// tc_mca_std_lib/POUs/ChangeConfig/FB_ReadParameterInNc_v1_00
///#########################################################
///Function block to read parameter in Nc.
///
///	Library:		
///	Tc2_MC2.lib
/// Tc2_System.lib
///
///	Global Variables:
///	
///	Data types:
///	
///	External functions:
///
///	History:
///	2014-02-05	v1.00	NB	Release code.
///
///	Known bugs:
///
///
///
///###########################################################
FUNCTION_BLOCK FB_ReadParameterInNc_v1_00
VAR_INPUT
	bExecute: BOOL;
	///16#4000=Axisdata, 16#5000=Encoderdata, 16#6000=Controldata, 16#7000=Drivedata
	nDeviceGroup: UDINT;
	nIndexOffset: UDINT;
END_VAR
VAR_OUTPUT
	nData: DWORD;
	bBusy: BOOL;
	bDone: BOOL;
	bError: BOOL;
	nErrorId: UDINT;
END_VAR
VAR_IN_OUT
	Axis: AXIS_REF;
END_VAR
VAR
	nState: UINT;
	fbADSREAD: ADSREAD;
END_VAR

(*Sequence to read parameter in Nc*)
CASE nState OF
0:  (*Start sequence. Wait until bExecute is TRUE*)
	IF bExecute THEN
		bBusy:=TRUE;
		bError:=FALSE;
		nErrorId:=0;
		nState:=10;
	END_IF

10: (*Read parameter in Nc*)
	fbADSREAD(
		PORT:=500,
		IDXGRP:=nDeviceGroup+Axis.NcToPlc.AxisId,
		IDXOFFS:=nIndexOffset,
		LEN:=SIZEOF(nData),
		DESTADDR:=ADR(nData),
		READ:=TRUE);

	(*Wait until it's done or if an error occurs*)
	IF NOT fbADSREAD.ERR THEN
		IF NOT fbADSREAD.BUSY THEN
			fbADSREAD(READ:=FALSE);
			nState:=20;
		END_IF
	ELSE
		nErrorId:=fbADSREAD.ERRID;
		nState:=999;
	END_IF

20: (*Sequense is done. Waits until bExecute is FALSE*)
	bBusy:=FALSE;
	bDone:=TRUE;
	IF NOT bExecute THEN
		bDone:=FALSE;
		nState:=0;
	END_IF

999: (*Error in sequence*)
	bError:=TRUE;
	bBusy:=FALSE;
	bDone:=FALSE;
	fbADSREAD(READ:=FALSE);
	IF NOT bExecute THEN
		nState:=0;
	END_IF

END_CASE

END_FUNCTION_BLOCK

// tc_mca_std_lib/POUs/Motion/Homing/FB_HomeWriteSoftLimEnable
FUNCTION_BLOCK FB_HomeWriteSoftLimEnable
VAR_INPUT
	En: BOOL;
	bReset: BOOL;
    bExecute: BOOL;		
	bSofLimEnableLow: BOOL:=TRUE;
	bSofLimEnableHigh: BOOL:=TRUE;
END_VAR
VAR_IN_OUT
	Axis: AXIS_REF;
END_VAR
VAR_OUTPUT
	EnO: BOOL;	
	bBusy: BOOL;
	bDone: BOOL;
	bError: BOOL;
	nErrorId: UDINT;	
END_VAR
VAR
	fbExecuteRiseEdge: R_TRIG;
	fbWriteSoftLimEnableLow:FB_WriteParameterInNc_v1_00;
	fbWriteSoftLimEnableHigh:FB_WriteParameterInNc_v1_00;
END_VAR

En:=EnO;
IF bReset THEN
	bError:=FALSE;
	nErrorId:=0;
END_IF 

fbExecuteRiseEdge(CLK:=bExecute);

fbWriteSoftLimEnableLow(
	bExecute:=bExecute,
	nDeviceGroup:= 16#5000,
	nIndexOffset:= 16#B,
	nData:=BOOL_TO_DWORD(bSofLimEnableLow),
	Axis:= Axis);
	
fbWriteSoftLimEnableHigh(
	bExecute:=bExecute,
	nDeviceGroup:= 16#5000,
	nIndexOffset:= 16#C,
	nData:=BOOL_TO_DWORD(bSofLimEnableHigh),
	Axis:= Axis);

bBusy:=fbWriteSoftLimEnableLow.bBusy OR fbWriteSoftLimEnableHigh.bBusy;
bDone:=fbWriteSoftLimEnableLow.bDone AND fbWriteSoftLimEnableHigh.bDone AND bExecute;

bError:=fbWriteSoftLimEnableHigh.bError OR fbWriteSoftLimEnableLow.bError;
IF fbWriteSoftLimEnableHigh.bError THEN
  nErrorId:=fbWriteSoftLimEnableHigh.nErrorId;
ELSIF fbWriteSoftLimEnableLow.bError THEN
  nErrorId:=fbWriteSoftLimEnableLow.nErrorId;
END_IF

END_FUNCTION_BLOCK

// tc_mca_std_lib/POUs/Motion/Homing/FB_HomeReadNcVelocities
FUNCTION_BLOCK FB_HomeReadNcVelocities
VAR_INPUT
	En: BOOL;
	bReset: BOOL;
    bExecute: BOOL;			
END_VAR
VAR_IN_OUT
	Axis: AXIS_REF;
END_VAR
VAR_OUTPUT
	EnO: BOOL;	
	bBusy: BOOL;
	bDone: BOOL;
	bError: BOOL;
	nErrorId: UDINT;	
	fVelocityToCam: LREAL;
	fVelocityFromCam: LREAL;
END_VAR
VAR
	fbReadVelocityToCam:FB_ReadFloatParameter;
	fbReadVelocityFromCam:FB_ReadFloatParameter;
END_VAR

En:=EnO;
IF bReset THEN
	bError:=FALSE;
	nErrorId:=0;
END_IF 
	
fbReadVelocityToCam(
	bExecute:=bExecute,
	nDeviceGroup:= 16#4000,
	nIndexOffset:= 16#6,
	Axis:= Axis);
	
fbReadVelocityFromCam(
	bExecute:=bExecute,
	nDeviceGroup:= 16#4000,
	nIndexOffset:= 16#7,
	Axis:= Axis);
	
fVelocityToCam:=fbReadVelocityToCam.nData;
fVelocityFromCam:=fbReadVelocityFromCam.nData;	

bBusy:=fbReadVelocityFromCam.bBusy OR fbReadVelocityToCam.bBusy;
bDone:=fbReadVelocityFromCam.bDone AND fbReadVelocityToCam.bDone AND bExecute;

bError:=fbReadVelocityToCam.bError OR fbReadVelocityFromCam.bError;
IF fbReadVelocityToCam.bError THEN
  nErrorId:=fbReadVelocityToCam.nErrorId;
ELSIF fbReadVelocityFromCam.bError THEN
  nErrorId:=fbReadVelocityFromCam.nErrorId;
END_IF

END_FUNCTION_BLOCK

// tc_mca_std_lib/POUs/ChangeConfig/FB_ReadFloatParameter
FUNCTION_BLOCK FB_ReadFloatParameter
VAR_INPUT
	bExecute: BOOL;
	///16#4000=Axisdata, 16#5000=Encoderdata, 16#6000=Controldata, 16#7000=Drivedata
	nDeviceGroup: UDINT;
	nIndexOffset: UDINT;
END_VAR
VAR_OUTPUT
	nData: LREAL;
	bBusy: BOOL;
	bDone: BOOL;
	bError: BOOL;
	nErrorId: UDINT;
END_VAR
VAR_IN_OUT
	Axis: AXIS_REF;
END_VAR
VAR
	nState: UINT;
	fbADSREAD: ADSREAD;
END_VAR

(*Sequence to read parameter in Nc*)
CASE nState OF
0:  (*Start sequence. Wait until bExecute is TRUE*)
	IF bExecute THEN
		bBusy:=TRUE;
		bError:=FALSE;
		nErrorId:=0;
		nState:=10;
	END_IF

10: (*Read parameter in Nc*)
	fbADSREAD(
		PORT:=500,
		IDXGRP:=nDeviceGroup+Axis.NcToPlc.AxisId,
		IDXOFFS:=nIndexOffset,
		LEN:=SIZEOF(nData),
		DESTADDR:=ADR(nData),
		READ:=TRUE);

	(*Wait until it's done or if an error occurs*)
	IF NOT fbADSREAD.ERR THEN
		IF NOT fbADSREAD.BUSY THEN
			fbADSREAD(READ:=FALSE);
			nState:=20;
		END_IF
	ELSE
		nErrorId:=fbADSREAD.ERRID;
		nState:=999;
	END_IF

20: (*Sequense is done. Waits until bExecute is FALSE*)
	bBusy:=FALSE;
	bDone:=TRUE;
	IF NOT bExecute THEN
		bDone:=FALSE;
		nState:=0;
	END_IF

999: (*Error in sequence*)
	bError:=TRUE;
	bBusy:=FALSE;
	bDone:=FALSE;
	fbADSREAD(READ:=FALSE);
	IF NOT bExecute THEN
		nState:=0;
	END_IF

END_CASE

END_FUNCTION_BLOCK

// tc_mca_std_lib/POUs/Motion/Homing/FB_HomeFinish
FUNCTION_BLOCK FB_HomeFinish
VAR_INPUT
	En: BOOL;
	bReset: BOOL;
    bExecute: BOOL;	
    nCmdData: UINT;
	bSofLimEnableLow: BOOL:=TRUE;
	bSofLimEnableHigh: BOOL:=TRUE;			
END_VAR
VAR_IN_OUT
	Axis: AXIS_REF;
END_VAR
VAR_OUTPUT
	EnO: BOOL;	
	bBusy: BOOL;
	bDone: BOOL;
	bError: BOOL;
	nErrorId: UDINT;
END_VAR
VAR		
	fbHomewriteSoftLimEnable:FB_HomeWriteSoftLimEnable;	
	fbExecuteRiseEdge: R_TRIG;	
	bExecuteWriteNC:BOOL:=FALSE;
	nState:INT:=0;
END_VAR

En:=EnO;
IF bReset THEN
	bError:=FALSE;
	nErrorId:=0;
END_IF 

IF NOT bExecute THEN
  bExecuteWriteNC:=FALSE;
  fbHomewriteSoftLimEnable.bSofLimEnableLow:=bSofLimEnableLow;
  fbHomewriteSoftLimEnable.bSofLimEnableHigh:=bSofLimEnableHigh;   
  nState:=0;
END_IF

fbExecuteRiseEdge(CLK:=bExecute);
IF fbExecuteRiseEdge.Q THEN
  bExecuteWriteNC:=TRUE;  
  fbHomewriteSoftLimEnable.bSofLimEnableLow:=bSofLimEnableLow;
  fbHomewriteSoftLimEnable.bSofLimEnableHigh:=bSofLimEnableHigh;
END_IF

// Write to NC (disable soft limits)
fbHomewriteSoftLimEnable(
	En:=En,
	bExecute:=bExecuteWriteNC AND bExecute,
	Axis:=Axis,
	bReset:=bReset,	
);

bBusy:=fbHomewriteSoftLimEnable.bBusy;
bDone:=fbHomewriteSoftLimEnable.bDone;

bError:=fbHomewriteSoftLimEnable.bError;
IF fbHomewriteSoftLimEnable.bError THEN
  nErrorId:=fbHomewriteSoftLimEnable.nErrorId;
END_IF

END_FUNCTION_BLOCK

// POUs/Motion/FB_MotionHoming
FUNCTION_BLOCK FB_MotionHoming
VAR_IN_OUT
    stMotionStage: ST_MotionStage;
END_VAR
VAR_INPUT
    bExecute: BOOL;
END_VAR
VAR_OUTPUT
    bBusy: BOOL;
    bDone: BOOL;
    bError: BOOL;
    nErrorID: UDINT;
END_VAR
VAR
    fbSetPos: MC_SetPosition;
    fbJog: MC_Jog;
    rtExec: R_TRIG;
    ftExec: F_TRIG;
    nHomeStateMachine: INT := IDLE;
    nStateAfterStop: INT;
    nMoves: INT;
    bFirstDirection: BOOL;
    bAtHome: BOOL;
    bMove: BOOL;
    nErrCount: INT;
    bInterrupted: BOOL;
END_VAR
VAR CONSTANT
    IDLE: INT := 0;
    NEXT_MOVE: INT := 1;
    CHECK_FWD: INT := 2;
    CHECK_BWD: INT := 3;
    FINAL_MOVE: INT := 4;
    FINAL_SETPOS: INT := 5;
    ERROR: INT := 6;
    WAIT_STOP: INT := 7;

    (*
        This is a simpler way of disabling the soft limits that ends up being really obvious if something has gone wrong.
        If you turn the limits off/on, not only do you need to keep track of if you had soft limits set,
        but you need to always restore this properly or risk some issue.
        Instead, I set position to a ridiculous value that can always move forward or backward.
        If this gets stuck for any reason it's very clear that something has gone wrong,
        rather than a silent failure of the soft limit marks.
    *)
    FWD_START: LREAL := -99999999;
    BWD_START: LREAL :=  99999999;
END_VAR


fbSetPos.Options.ClearPositionLag := TRUE;
rtExec(CLK:=bExecute);
ftExec(CLK:=bExecute);

bError R= NOT bExecute;
IF NOT bError THEN
    nErrorID := 0;
END_IF

CASE stMotionStage.nHomingMode OF
    E_EpicsHomeCmd.LOW_LIMIT:
        bFirstDirection := FALSE;
        bAtHome := NOT stMotionStage.bLimitBackwardEnable;
        bMove := TRUE;
    E_EpicsHomeCmd.HIGH_LIMIT:
        bFirstDirection := TRUE;
        bAtHome := NOT stMotionStage.bLimitForwardEnable;
        bMove := TRUE;
    E_EpicsHomeCmd.HOME_VIA_LOW:
        bFirstDirection := FALSE;
        bAtHome := stMotionStage.bHome;
        bMove := TRUE;
    E_EpicsHomeCmd.HOME_VIA_HIGH:
        bFirstDirection := TRUE;
        bAtHome := stMotionStage.bHome;
        bMove := TRUE;
    E_EpicsHomeCmd.ABSOLUTE_SET:
        fbSetPos(
            Axis:=stMotionStage.Axis,
            Execute:=bExecute,
            Position:=stMotionStage.fHomePosition);
        bBusy := rtExec.Q;
        bDone := NOT rtExec.Q;
        bMove := FALSE;
    E_EpicsHomeCmd.NONE:
        bMove := FALSE;
        bBusy := rtExec.Q;
        bDone := NOT rtExec.Q;
    ELSE
        bMove := FALSE;
END_CASE

IF bMove THEN
    IF bBusy AND ftExec.Q THEN
        nHomeStateMachine := ERROR;
        bInterrupted := TRUE;
    END_IF
    CASE nHomeStateMachine OF
        // Wait for a rising edge
        IDLE:
            bBusy := FALSE;
            nErrCount := 0;
            fbSetPos(
                Axis:=stMotionStage.Axis,
                Execute:=FALSE);
            fbJog(
                Axis:=stMotionStage.Axis,
                JogForward:=FALSE,
                JogBackwards:=FALSE);
            IF rtExec.Q THEN
                nHomeStateMachine := NEXT_MOVE;
                nMoves := 0;
                bDone := FALSE;
                bBusy := TRUE;
                bError := FALSE;
                nErrorID := 0;
                bInterrupted := FALSE;
            END_IF
        // Figure out whether to move forward, move backward, or give up
        NEXT_MOVE:
            fbSetPos(
                Axis:=stMotionStage.Axis,
                Execute:=FALSE);
            fbJog(
                Axis:=stMotionStage.Axis,
                JogForward:=FALSE,
                JogBackwards:=FALSE);
            CASE nMoves OF
                0:
                    IF bFirstDirection THEN
                        nStateAfterStop := CHECK_FWD;
                    ELSE
                        nStateAfterStop := CHECK_BWD;
                    END_IF
                1:
                    IF NOT bFirstDirection THEN
                        nStateAfterStop := CHECK_FWD;
                    ELSE
                        nStateAfterStop := CHECK_BWD;
                    END_IF
                ELSE
                    nStateAfterStop := ERROR;
            END_CASE
            nMoves := nMoves + 1;
            IF bAtHome THEN
                nStateAfterStop := FINAL_MOVE;
            END_IF
            nHomeStateMachine := WAIT_STOP;
        // Move forward until we find the home signal or reach end of travel
        CHECK_FWD:
            fbSetPos(
                Axis:=stMotionStage.Axis,
                Execute:=TRUE,
                Position:=FWD_START);
            fbJog(
                Axis:=stMotionStage.Axis,
                JogForward:=stMotionStage.bLimitForwardEnable AND NOT bATHome,
                JogBackwards:=FALSE,
                Mode:=E_JogMode.MC_JOGMODE_CONTINOUS,
                Velocity:=stMotionStage.stAxisParameters.fRefVeloSearch);
            IF NOT fbJog.JogForward THEN
                nHomeStateMachine := NEXT_MOVE;
            ELSIF fbJog.Error THEN
                fbJog(
                    Axis:=stMotionStage.Axis,
                    JogForward:=FALSE,
                    JogBackwards:=FALSE);
                nErrCount := nErrCount + 1;
                IF nErrCount >= 3 THEN
                    nHomeStateMachine := ERROR;
                END_IF
            END_IF
        // Move backward until we find the home signal or reach end of travel
        CHECK_BWD:
            fbSetPos(
                Axis:=stMotionStage.Axis,
                Execute:=TRUE,
                Position:=BWD_START);
            fbJog(
                Axis:=stMotionStage.Axis,
                JogForward:=FALSE,
                JogBackwards:=stMotionStage.bLimitBackwardEnable AND NOT bATHome,
                Mode:=E_JogMode.MC_JOGMODE_CONTINOUS,
                Velocity:=stMotionStage.stAxisParameters.fRefVeloSearch);
            IF NOT fbJog.JogBackwards THEN
                nHomeStateMachine := NEXT_MOVE;
            ELSIF fbJog.Error THEN
                fbJog(
                    Axis:=stMotionStage.Axis,
                    JogForward:=FALSE,
                    JogBackwards:=FALSE);
                nErrCount := nErrCount + 1;
                IF nErrCount >= 3 THEN
                    nHomeStateMachine := ERROR;
                END_IF
            END_IF
        // Set position to get within soft lims, move slowly off signal
        FINAL_MOVE:
            fbSetPos(
                Axis:=stMotionStage.Axis,
                Execute:=TRUE,
                Position:=stMotionStage.fHomePosition);
            IF bAtHome THEN
                fbJog(
                    Axis:=stMotionStage.Axis,
                    JogForward:=NOT bFirstDirection,
                    JogBackwards:=bFirstDirection,
                    Mode:=E_JogMode.MC_JOGMODE_CONTINOUS,
                    Velocity:=stMotionStage.stAxisParameters.fRefVeloSync);
            ELSIF fbJog.Error THEN
                fbJog(
                    Axis:=stMotionStage.Axis,
                    JogForward:=FALSE,
                    JogBackwards:=FALSE);
                nErrCount := nErrCount + 1;
                IF nErrCount >= 3 THEN
                    nHomeStateMachine := ERROR;
                END_IF
            ELSE
                fbJog(
                    Axis:=stMotionStage.Axis,
                    JogForward:=FALSE,
                    JogBackwards:=FALSE);
                fbSetPos(
                    Axis:=stMotionStage.Axis,
                    Execute:=FALSE);
                nHomeStateMachine := WAIT_STOP;
                nStateAfterStop := FINAL_SETPOS;
            END_IF
        FINAL_SETPOS:
            fbSetPos(
                Axis:=stMotionStage.Axis,
                Execute:=TRUE,
                Position:=stMotionStage.fHomePosition);
            nHomeStateMachine := IDLE;
            bBusy := FALSE;
            bDone := TRUE;
        ERROR:
            bError := TRUE;
            nErrorID := fbJog.ErrorID;
            nHomeStateMachine := FINAL_SETPOS;
            fbSetPos(
                Axis:=stMotionStage.Axis,
                Execute:=FALSE);
            IF bInterrupted THEN
                stMotionStage.sCustomErrorMessage := 'Homing interrupted';
            ELSE
                stMotionStage.sCustomErrorMessage := 'Homing failure';
            END_IF
        WAIT_STOP:
            IF stMotionStage.Axis.Status.NotMoving THEN
                nHomeStateMachine := nStateAfterStop;
            END_IF
    END_CASE
END_IF

END_FUNCTION_BLOCK

// POUs/Motion/FB_EncSaveRestore
FUNCTION_BLOCK FB_EncSaveRestore
VAR_IN_OUT
    stMotionStage: ST_MotionStage;
END_VAR
VAR_INPUT
    bEnable: BOOL;
END_VAR
VAR_OUTPUT
END_VAR
VAR
    fbSetPos: MC_SetPosition;
    timer: TON;
    bInit: BOOL;
    bLoad: BOOL;
    nLatchError: UDINT;
    bEncError: BOOL;
    tRetryDelay: TIME := T#1s;
    nMaxRetries: UINT := 10;
    nCurrTries: UINT := 0;
    bWaitRetry: BOOL;
    tonRetry: TON;
END_VAR
VAR PERSISTENT
    bSaved: BOOL;
    fPosition: LREAL;
END_VAR

IF bEnable THEN
    // Trigger a load if anything was saved at all
    IF NOT bInit THEN
        bInit := TRUE;
        bLoad S= bSaved;
        fbSetPos.Options.ClearPositionLag := TRUE;
    END_IF

    // Set our position if bLoad is true
    fbSetPos(
        Axis:=stMotionStage.Axis,
        Execute:=bLoad,
        Position:=fPosition);

    // Only load once, at startup
    bLoad R= fbSetPos.Done OR fbSetPos.Error;

    IF fbSetPos.Error THEN
        // Keep the error latched, it can disappear if Execute is set to FALSE
        nLatchError := fbSetPos.ErrorID;
        nCurrTries := nCurrTries + 1;
        IF nCurrTries >= nMaxRetries THEN
            // Alert the user that something has gone wrong
            stMotionStage.bError := TRUE;
            stMotionStage.nErrorId := nLatchError;
            stMotionStage.sCustomErrorMessage := 'Error loading previously saved position.';
        ELSE
            // Reset the FB for the next retry
            fbSetPos(
                Axis:=stMotionStage.Axis,
                Execute:=FALSE,
                Position:=fPosition);
            // Try again
            bWaitRetry := TRUE;
        END_IF
    END_IF

    tonRetry(
        IN := bWaitRetry,
        PT := tRetryDelay);

    bLoad S= tonRetry.Q;
    bWaitRetry R= tonRetry.Q;

    // Check ST_MotionStage for an encoder error (range 0x44nn)
    bEncError := stMotionStage.bError AND stMotionStage.nErrorId >= 16#4400 AND stMotionStage.nErrorId <= 16#44FF;

    // Do not save if we're currently loading or if there is an encoder error
    IF NOT bLoad AND NOT bEncError AND NOT bWaitRetry THEN
        fPosition := stMotionStage.stAxisStatus.fActPosition;
        // This persistent variable lets us check if anything was saved
        // It will be TRUE at startup if we have saved values
        bSaved := TRUE;
    END_IF
END_IF

END_FUNCTION_BLOCK

// POUs/Motion/FB_LogMotionError
FUNCTION_BLOCK FB_LogMotionError
(*
    If the motion struct has an error, log it.

    The log condition is:
    - When bError goes TRUE (catch transition from no error to error)
    - When the error message changes while bError is TRUE (catch transition from error a to error b)

    Includes the motor name and the NC error id in the json blob
*)
VAR_IN_OUT
    stMotionStage: ST_MotionStage;
END_VAR
VAR_INPUT
    bEnable: BOOL;
END_VAR
VAR
    fbLogMessage: FB_LogMessage;
    rtNewError: R_TRIG;
    bChangedError: BOOL;
    sPrevErr: STRING;
    fbJson: FB_JsonSaxWriter;
END_VAR


rtNewError(CLK:=stMotionStage.bError);
bChangedError := stMotionStage.sErrorMessage <> '' AND stMotionStage.sErrorMessage <> sPrevErr;
sPrevErr := stMotionStage.sErrorMessage;

IF bEnable AND (rtNewError.Q OR bChangedError) THEN
    fbJson.StartObject();
    fbJson.AddKey('schema');
    fbJson.AddString('ST_MotionStage.bError');
    fbJson.AddKey('dut_name');
    fbJson.AddString(stMotionStage.sName);
    fbJson.AddKey('axis_name');
    fbJson.AddString(stMotionStage.stAxisParameters.sAxisName);
    fbJson.AddKey('axis_id');
    fbJson.AddUdint(stMotionStage.stAxisParameters.AxisId);
    fbJson.AddKey('err_id');
    fbJson.AddUdint(stMotionStage.nErrorId);
    fbJson.AddKey('position');
    fbJson.AddLreal(stMotionStage.stAxisStatus.fActPosition);
    fbJson.AddKey('position_lag');
    fbJson.AddLreal(stMotionStage.stAxisStatus.fActDiff);
    fbJson.EndObject();
    fbLogMessage.sJson := fbJson.GetDocument();
    fbLogMessage(
        sMsg := stMotionStage.sErrorMessage,
        eSevr := TcEventSeverity.Error,
        eSubsystem := E_Subsystem.MOTION,
    );
    fbJson.ResetDocument();
END_IF

END_FUNCTION_BLOCK

// POUs/Motion/Utils/FB_SetEnables
FUNCTION_BLOCK FB_SetEnables
// Update the all enable booleans based on the booleans that make them up
VAR_IN_OUT
    stMotionStage: ST_MotionStage;
END_VAR

stMotionStage.bAllForwardEnable := stMotionStage.bLimitForwardEnable AND (stMotionStage.bGantryForwardEnable OR NOT stMotionStage.bGantryAxis) AND stMotionStage.stEPSForwardEnable.bEPS_OK;
stMotionStage.bAllBackwardEnable := stMotionStage.bLimitBackwardEnable AND (stMotionStage.bGantryBackwardEnable OR NOT stMotionStage.bGantryAxis) AND stMotionStage.stEPSBackwardEnable.bEPS_OK;

stMotionStage.bAllEnable := stMotionStage.bEnable AND stMotionStage.bHardwareEnable AND stMotionStage.stEPSPowerEnable.bEPS_OK;
stMotionStage.bAllEnable R= NOT stMotionStage.bUserEnable;

END_FUNCTION_BLOCK

// POUs/Motion/FB_EncoderValue
FUNCTION_BLOCK FB_EncoderValue
(*
    Process the encoder value for ST_MotionStage

    A few different problems this is trying to solve:
        1. Different encoders show as different types in the IO,
           but we want a consistent type for checks and for PVs
        2. Some inverted encoders display as very high numbers
           as they count down from max int instead of up from 0
        3. Some encoders have raw signed values, others unsigned.

    To this end, we figure out which encoder is linked and process
    the value appropriately.
*)
VAR_IN_OUT
    stMotionStage: ST_MotionStage;
END_VAR

IF stMotionStage.nRawEncoderULINT <> 0 THEN
    IF stMotionStage.nRawEncoderULINT < 4294967296 THEN
        stMotionStage.nEncoderCount := ULINT_TO_UDINT(stMotionStage.nRawEncoderULINT);
    ELSE
        stMotionStage.nEncoderCount := ULINT_TO_UDINT(18446744073709551615 - stMotionStage.nRawEncoderULINT);
    END_IF
ELSIF stMotionStage.nRawEncoderUINT <> 0 THEN
    stMotionStage.nEncoderCount := UINT_TO_UDINT(stMotionStage.nRawEncoderUINT);
ELSIF stMotionStage.nRawEncoderINT <> 0 THEN
    stMotionStage.nEncoderCount := INT_TO_UDINT(stMotionStage.nRawEncoderINT);
ELSE
    stMotionStage.nEncoderCount := 0;
END_IF

END_FUNCTION_BLOCK

// POUs/Motion/FB_MotionStageNCParams
FUNCTION_BLOCK FB_MotionStageNCParams
(*
    Read and refresh axis parameters struct on ST_MotionStage
*)
VAR_IN_OUT
    stMotionStage: ST_MotionStage;
END_VAR
VAR_INPUT
    bEnable: BOOL;
    tRefreshDelay: TIME;
END_VAR
VAR_OUTPUT
    bError: BOOL;
END_VAR
VAR
    mcReadParams: MC_ReadParameterSet;
    timer: TON;
    bExecute: BOOL := TRUE;
    nLatchErrId: UDINT;
END_VAR

timer(
    IN:=bEnable AND NOT bExecute,
    PT:=tRefreshDelay);
bExecute S= timer.Q;
mcReadParams(
    Parameter:=stMotionStage.stAxisParameters,
    Axis:=stMotionStage.Axis,
    Execute:=bEnable AND bExecute,
    Error=>bError);
IF mcReadParams.ErrorID <> 0 THEN
    nLatchErrId := 0;
END_IF
bExecute R= mcReadParams.Done OR mcReadParams.Error;
stMotionStage.bAxisParamsInit S= mcReadParams.Done;

END_FUNCTION_BLOCK

// POUs/Motion/States/FB_PositionStateND_Core
FUNCTION_BLOCK FB_PositionStateND_Core
(*
    Collection of all the actions shared between all states FBs
    This is used in e.g.
    - FB_PositionState1D
    - FB_PositionState2D
    - ... etc.
    - FB_PositionStatePMPS1D
    - FB_PositionStatePMPS2D
    - ... etc.

    This is essentially input handling, position state reading, standard management blocks, and the motion state machine.
*)
VAR_IN_OUT
    // All motors to be used in the states move, including blank/uninitialized structs.
    astMotionStageMax: ARRAY[1..MotionConstants.MAX_STATE_MOTORS] OF ST_MotionStage;
    // All position states for all motors, including unused/invalid states.
    astPositionStateMax: ARRAY[1..MotionConstants.MAX_STATE_MOTORS] OF ARRAY[1..GeneralConstants.MAX_STATES] OF ST_PositionState;
    // Normal EPICS inputs, gathered into a single struct
    stEpicsToPlc: ST_StateEpicsToPlc;
    // Normal EPICS outputs, gathered into a single struct
    stPlcToEpics: ST_StatePlcToEpics;
    // Set this to a nonzero value to request a new move. It will be reset to zero every cycle. This should be hooked up to a user's EPICS enum input.
    eEnumSet: UINT;
    // The current state index, or zero if we are not at a state. This should be hooked up to a user's EPICS enum output.
    eEnumGet: UINT;
END_VAR
VAR_INPUT
    // Set this to TRUE to enable input state moves, or FALSE to disable them.
    bEnable: BOOL;
    // Set this to the number of motors to be included in astMotionStageMax
    nActiveMotorCount: UINT;
END_VAR
VAR_OUTPUT
    // The current position index goal, where the motors are supposed to be moving towards.
    nCurrGoal: UINT;
END_VAR
VAR
    fbInput: FB_StatesInputHandler;
    fbInternal: FB_PositionStateInternalND;
    fbMove: FB_PositionStateMoveND;
    fbRead: FB_PositionStateReadND;
    astMoveGoals: ARRAY[1..MotionConstants.MAX_STATE_MOTORS] OF ST_PositionState;
    stInvalidPos: ST_PositionState;
    nIterMotor: DINT;
END_VAR


stEpicsToPlc.nSetValue := eEnumSet;

fbRead(
    astMotionStage:=astMotionStageMax,
    astPositionState:=astPositionStateMax,
    nActiveMotorCount:=nActiveMotorCount,
    bKnownState=>,
    bMovingState=>,
    nPositionIndex=>stPlcToEpics.nGetValue,
);

fbInput(
    stUserInput:=stEpicsToPlc,
    bMoveBusy:=fbMove.bBusy,
    nStartingState:=fbRead.nPositionIndex,
    nCurrGoal=>nCurrGoal,
    bExecMove=>,
    bResetMove=>,
);

fbInternal(
    astMotionStage:=astMotionStageMax,
    astPositionState:=astPositionStateMax,
);

FOR nIterMotor := 1 TO MotionConstants.MAX_STATE_MOTORS DO
    IF nCurrGoal > 0 THEN
        astMoveGoals[nIterMotor] := astPositionStateMax[nIterMotor][nCurrGoal];
    ELSE
        astMoveGoals[nIterMotor] := stInvalidPos;
    END_IF
END_FOR

fbMove(
    astMotionStage:=astMotionStageMax,
    astPositionState:=astMoveGoals,
    nActiveMotorCount:=nActiveMotorCount,
    bExecute:=fbInput.bExecMove AND bEnable,
    bReset:=fbInput.bResetMove,
    enumMotionRequest:=E_MotionRequest.INTERRUPT,
    bAtState=>,
    bError=>stPlcToEpics.bError,
    nErrorID=>stPlcToEpics.nErrorID,
    sErrorMessage=>stPlcToEpics.sErrorMsg,
    bBusy=>stPlcToEpics.bBusy,
    bDone=>stPlcToEpics.bDone,
);

eEnumSet := stEpicsToPlc.nSetValue;
eEnumGet := stPlcToEpics.nGetValue;

END_FUNCTION_BLOCK

// POUs/Motion/States/FB_PositionState2D
FUNCTION_BLOCK FB_PositionState2D
(*
    2-Dimensional position state function block.

    This allows the user to move 2 motors among some set of named state positions.

    To use a states block, you must define enums that match the state options and give them pytmc pragmas.
    See FB_PositionState1D_InOut for a simple example.
    These enums must be passed in as the eEnumSet and eEnumGet VAR_IN_OUT variables.
    The enum values must match the array indices in astPositionState1 and astPositionState2.

    A move will begin when eEnumSet is set to a positive, nonzero value. eEnumSet will be reset to 0 on every cycle, allowing us
    to accept a new, possibly conflicting, move request on the next cycle to interrupt the first.

    The motors must already be set up for point-to-point motion via FB_MotionStage, etc., for this function block to work properly.

    With no PMPS handling, this FB basically just links the state names with positions in both directions for set and readback.
*)
VAR_IN_OUT
    // The 1st motor to move
    stMotionStage1: ST_MotionStage;
    // The 2nd motor to move
    stMotionStage2: ST_MotionStage;
    // All possible position states for motor 1, including unused/invalid states.
    {attribute 'pytmc' := '
        pv: STATE:01
        io: io
        expand: :%.2d
    '}
    astPositionState1: ARRAY[1..GeneralConstants.MAX_STATES] OF ST_PositionState;
    // All possible position states for motor 2, including unused/invalid states.
    {attribute 'pytmc' := '
        pv: STATE:02
        io: io
        expand: :%.2d
    '}
    astPositionState2: ARRAY[1..GeneralConstants.MAX_STATES] OF ST_PositionState;
    // Set this to a nonzero value to request a new move. It will be reset to zero every cycle. This should be hooked up to a user's EPICS enum input.
    eEnumSet: UINT;
    // The current state index, or zero if we are not at a state. This should be hooked up to a user's EPICS enum output.
    eEnumGet: UINT;
END_VAR
VAR_INPUT
    // Set this to TRUE to enable input state moves, or FALSE to disable them.
    bEnable: BOOL;
    // Normal EPICS inputs, gathered into a single struct
    {attribute 'pytmc' := 'pv: STATE'}
    stEpicsToPlc: ST_StateEpicsToPlc;
END_VAR
VAR_OUTPUT
    // Normal EPICS outputs, gathered into a single struct
    {attribute 'pytmc' := 'pv: STATE'}
    stPlcToEpics: ST_StatePlcToEpics;
END_VAR
VAR
    fbCore: FB_PositionStateND_Core;
    astMotionStageMax: ARRAY[1..MotionConstants.MAX_STATE_MOTORS] OF ST_MotionStage;
    astPositionStateMax: ARRAY[1..MotionConstants.MAX_STATE_MOTORS] OF ARRAY[1..GeneralConstants.MAX_STATES] OF ST_PositionState;
END_VAR


astMotionStageMax[1] := stMotionStage1;
astMotionStageMax[2] := stMotionStage2;
astPositionStateMax[1] := astPositionState1;
astPositionStateMax[2] := astPositionState2;

fbCore(
    astMotionStageMax:=astMotionStageMax,
    astPositionStateMax:=astPositionStateMax,
    stEpicsToPlc:=stEpicsToPlc,
    stPlcToEpics:=stPlcToEpics,
    eEnumSet:=eEnumSet,
    eEnumGet:=eEnumGet,
    bEnable:=bEnable,
    nActiveMotorCount:=2,
);

stMotionStage1 := astMotionStageMax[1];
stMotionStage2 := astMotionStageMax[2];
astPositionState1 := astPositionStateMax[1];
astPositionState2 := astPositionStateMax[2];

END_FUNCTION_BLOCK

// POUs/Motion/PMPS/FB_PositionStatePMPS1D
FUNCTION_BLOCK FB_PositionStatePMPS1D
(*
    1-Dimensional position state function block with PMPS.

    This allows the user to move a motor among some set of named state positions with PMPS protection.

    To use a states block, you must define enums that match the state options and give them pytmc pragmas.
    See FB_PositionState1D_InOut for a simple example.
    These enums must be passed in as the eEnumSet and eEnumGet VAR_IN_OUT variables.
    The enum values must match the array indices in astPositionState.

    A move will begin when eEnumSet is set to a positive, nonzero value. eEnumSet will be reset to 0 on every cycle, allowing us
    to accept a new, possibly conflicting, move request on the next cycle to interrupt the first.

    The motor must already be set up for point-to-point motion via FB_MotionStage, etc., for this function block to work properly.

    PMPS handling is done via database lookups by setting sPmpsState on each position state and on
    the transition state input appropriately.
*)
VAR_IN_OUT
    // The motor to move.
    stMotionStage: ST_MotionStage;
    // All possible position states, including unused/invalid states.
    {attribute 'pytmc' := '
        pv: STATE
        io: io
        expand: :%.2d
    '}
    astPositionState: ARRAY[1..GeneralConstants.MAX_STATES] OF ST_PositionState;
    // Set this to a nonzero value to request a new move. It will be reset to zero every cycle. This should be hooked up to a user's EPICS enum input.
    eEnumSet: UINT;
    // The current state index, or zero if we are not at a state. This should be hooked up to a user's EPICS enum output.
    eEnumGet: UINT;
    // The fast fault output to fault to.
    fbFFHWO: FB_HardwareFFOutput;
    // The arbiter to request beam conditions from.
    fbArbiter: FB_Arbiter;
END_VAR
VAR_INPUT
    // Set this to TRUE to enable input state moves, or FALSE to disable them.
    bEnableMotion: BOOL;
    // Set this to TRUE to enable beam parameter checks, or FALSE to disable them.
    bEnableBeamParams: BOOL;
    // Set this to TRUE to enable position limit checks, or FALSE to disable them.
    bEnablePositionLimits: BOOL;
    // The name of the device for use in the PMPS DB lookup and diagnostic screens.
    sDeviceName: STRING;
    // The name of the transition state in the PMPS database.
    sTransitionKey: STRING;
    // Normal EPICS inputs, gathered into a single struct
    {attribute 'pytmc' := 'pv: STATE'}
    stEpicsToPlc: ST_StateEpicsToPlc;
    // PMPS EPICS inputs, gathered into a single struct
    {attribute 'pytmc' := 'pv: STATE'}
    stPMPSEpicsToPlc: ST_StatePMPSEpicsToPlc;
    // Set this to TRUE to re-read the loaded database immediately (useful for debug)
    bReadDBNow: BOOL;
END_VAR
VAR_OUTPUT
    // Normal EPICS outputs, gathered into a single struct
    {attribute 'pytmc' := 'pv: STATE'}
    stPlcToEpics: ST_StatePlcToEpics;
    // PMPS EPICS outputs, gathered into a single struct
    {attribute 'pytmc' := 'pv: STATE'}
    stPMPSPlcToEpics: ST_StatePMPSPlcToEpics;
    // The PMPS database lookup associated with the current position state.
    stDbStateParams: ST_DbStateParams;
END_VAR
VAR
    fbCore: FB_PositionStateND_Core;
    fbPMPSCore: FB_PositionStatePMPSND_Core;
    astMotionStageMax: ARRAY[1..MotionConstants.MAX_STATE_MOTORS] OF ST_MotionStage;
    astPositionStateMax: ARRAY[1..MotionConstants.MAX_STATE_MOTORS] OF ARRAY[1..GeneralConstants.MAX_STATES] OF ST_PositionState;
END_VAR


astMotionStageMax[1] := stMotionStage;
astPositionStateMax[1] := astPositionState;

fbCore(
    astMotionStageMax:=astMotionStageMax,
    astPositionStateMax:=astPositionStateMax,
    stEpicsToPlc:=stEpicsToPlc,
    stPlcToEpics:=stPlcToEpics,
    eEnumSet:=eEnumSet,
    eEnumGet:=eEnumGet,
    bEnable:=bEnableMotion,
    nActiveMotorCount:=1,
    nCurrGoal=>,
);
fbPMPSCore(
    astMotionStageMax:=astMotionStageMax,
    astPositionStateMax:=astPositionStateMax,
    stEpicsToPlc:=stEpicsToPlc,
    stPMPSEpicsToPlc:=stPMPSEpicsToPlc,
    stPlcToEpics:=stPlcToEpics,
    stPMPSPlcToEpics:=stPMPSPlcToEpics,
    fbFFHWO:=fbFFHWO,
    fbArbiter:=fbArbiter,
    bEnableBeamParams:=bEnableBeamParams,
    bEnablePositionLimits:=bEnablePositionLimits,
    nActiveMotorCount:=1,
    sDeviceName:=sDeviceName,
    sTransitionKey:=sTransitionKey,
    nCurrGoal:=fbCore.nCurrGoal,
    bReadDBNow:=bReadDBNow,
    stDbStateParams=>stDbStateParams,
);

stMotionStage := astMotionStageMax[1];
astPositionState := astPositionStateMax[1];

END_FUNCTION_BLOCK

// POUs/Motion/PMPS/FB_PositionStatePMPSND_Core
FUNCTION_BLOCK FB_PositionStatePMPSND_Core
(*
    Collection of all core actions shared between all PMPS states FBs
    This is used in e.g.
    - FB_PositionStatePMPS1D
    - FB_PositionStatePMPS2D
    - ... etc.

    This handles database reading, BPTM, motor enables, virtual limits, and all FFOS.
*)
VAR_IN_OUT
    // All motors to be used in the states move, including blank/uninitialized structs.
    astMotionStageMax: ARRAY[1..MotionConstants.MAX_STATE_MOTORS] OF ST_MotionStage;
    // All position states for all motors, including unused/invalid states.
    astPositionStateMax: ARRAY[1..MotionConstants.MAX_STATE_MOTORS] OF ARRAY[1..GeneralConstants.MAX_STATES] OF ST_PositionState;
    // Normal EPICS inputs, gathered into a single struct
    stEpicsToPlc: ST_StateEpicsToPlc;
    // PMPS EPICS inputs, gathered into a single struct
    stPMPSEpicsToPlc: ST_StatePMPSEpicsToPlc;
    // Normal EPICS outputs, gathered into a single struct
    stPlcToEpics: ST_StatePlcToEpics;
    // PMPS EPICS outputs, gathered into a single struct
    stPMPSPlcToEpics: ST_StatePMPSPlcToEpics;
    // The fast fault output to fault to.
    fbFFHWO: FB_HardwareFFOutput;
    // The arbiter to request beam conditions from.
    fbArbiter: FB_Arbiter;
END_VAR
VAR_INPUT
    // Set this to TRUE to enable beam parameter checks, or FALSE to disable them.
    bEnableBeamParams: BOOL;
    // Set this to TRUE to enable position limit checks, or FALSE to disable them.
    bEnablePositionLimits: BOOL;
    // Set this to the number of motors to be included in astMotionStageMax
    nActiveMotorCount: UINT;
    // The name of the device for use in the PMPS DB lookup and diagnostic screens.
    sDeviceName: STRING;
    // The name of the transition state in the PMPS database.
    sTransitionKey: STRING;
    // The current position index goal, where the motors are supposed to be moving towards.
    nCurrGoal: UINT;
    // Set this to TRUE to re-read the loaded database immediately (useful for debug)
    bReadDBNow: BOOL;
END_VAR
VAR_OUTPUT
    // The PMPS database lookup associated with the current position state.
    stDbStateParams: ST_DbStateParams;
END_VAR
VAR
    fbMotionReadPMPSDB: FB_MotionReadPMPSDBND;
    fbMotionBPTM: FB_MotionBPTM;
    fbMotionClearAsserts: FB_MotionClearAsserts;
    fbStatePMPSEnables: FB_StatePMPSEnablesND;
    fbMiscStatesErrorFFO: FB_MiscStatesErrorFFO;
    fbPerMotorFFO: FB_PerMotorFFOND;

    eStatePMPSStatus: E_StatePMPSStatus;
END_VAR


IF stPMPSEpicsToPlc.bMaintMode OR NOT stPMPSEpicsToPlc.bArbiterEnabled THEN
    eStatePMPSStatus := E_StatePMPSStatus.DISABLED;
ELSIF stPlcToEpics.nGetValue = 0 AND nCurrGoal = 0 THEN
    eStatePMPSStatus := E_StatePMPSStatus.UNKNOWN;
ELSIF stPlcToEpics.nGetValue = nCurrGoal THEN
    eStatePMPSStatus := E_StatePMPSStatus.AT_STATE;
ELSE
    eStatePMPSStatus := E_StatePMPSStatus.TRANSITION;
END_IF

fbMotionReadPMPSDB(
    astPositionState:=astPositionStateMax,
    fbFFHWO:=fbFFHWO,
    sTransitionKey:=sTransitionKey,
    sDeviceName:=sDeviceName,
    bReadNow:=bReadDBNow,
    astDbStateParams=>,
    bError=>,
);

fbMotionBPTM(
    astMotionStage:=astMotionStageMax,
    fbArbiter:=fbArbiter,
    fbFFHWO:=fbFFHWO,
    stGoalParams:=fbMotionReadPMPSDB.astDbStateParams[nCurrGoal],
    stTransParams:=fbMotionReadPMPSDB.astDbStateParams[0],
    nActiveMotorCount:=nActiveMotorCount,
    bEnable:=stPMPSEpicsToPlc.bArbiterEnabled AND bEnableBeamParams,
    bAtState:=stPlcToEpics.nGetValue = nCurrGoal AND nCurrGoal <> 0,
    sDeviceName:=sDeviceName,
    bTransitionAuthorized=>,
    bDone=>,
    bMotorCountError=>,
);

fbMotionClearAsserts(
    astDbStateParams:=fbMotionReadPMPSDB.astDbStateParams,
    fbArbiter:=fbArbiter,
    bExecute:=NOT fbMotionBPTM.bEnable,
);

fbStatePMPSEnables(
    astMotionStage:=astMotionStageMax,
    astPositionState:=astPositionStateMax,
    fbFFHWO:=fbFFHWO,
    bEnable:=bEnablePositionLimits,
    nActiveMotorCount:=nActiveMotorCount,
    nGoalStateIndex:=nCurrGoal,
    sDeviceName:=sDeviceName,
    bMaintMode:=stPMPSEpicsToPlc.bMaintMode,
    eStatePMPSStatus:=eStatePMPSStatus,
    bTransitionAuthorized:=fbMotionBPTM.bTransitionAuthorized,
    abEnabled=>,
    abForwardEnabled=>,
    abBackwardEnabled=>,
    abValidGoal=>,
    bMotorCountError=>,
);

IF bEnableBeamParams THEN
    fbMiscStatesErrorFFO.stCurrentBeamReq := fbMotionReadPMPSDB.astDbStateParams[stPlcToEpics.nGetValue].stBeamParams;
ELSE
    fbMiscStatesErrorFFO.stCurrentBeamReq := PMPS_GVL.cstFullBeam;
END_IF
fbMiscStatesErrorFFO(
    fbArbiter:=fbArbiter,
    fbFFHWO:=fbFFHWO,
    sDeviceName:=sDeviceName,
    bKnownState:=stPlcToEpics.nGetValue > 0,
    nTransitionID:=fbMotionReadPMPSDB.astDbStateParams[0].nRequestAssertionID,
);

fbPerMotorFFO(
    astMotionStage:=astMotionStageMax,
    fbFFHWO:=fbFFHWO,
    nActiveMotorCount:=nActiveMotorCount,
    sDeviceName:=sDeviceName,
    bMotorCountError=>,
);

stPMPSPlcToEpics.stTransitionDb := fbMotionReadPMPSDB.astDbStateParams[0];
stDbStateParams := fbMotionReadPMPSDB.astDbStateParams[stPlcToEpics.nGetValue];

END_FUNCTION_BLOCK

// POUs/Motion/PMPS/FB_PositionStatePMPS2D
FUNCTION_BLOCK FB_PositionStatePMPS2D
(*
    2-Dimensional position state function block with PMPS.

    This allows the user to move 2 motors among some set of named state positions with PMPS protection.

    To use a states block, you must define enums that match the state options and give them pytmc pragmas.
    See FB_PositionState1D_InOut for a simple example.
    These enums must be passed in as the eEnumSet and eEnumGet VAR_IN_OUT variables.
    The enum values must match the array indices in astPositionState1 and astPositionState2.

    A move will begin when eEnumSet is set to a positive, nonzero value. eEnumSet will be reset to 0 on every cycle, allowing us
    to accept a new, possibly conflicting, move request on the next cycle to interrupt the first.

    The motors must already be set up for point-to-point motion via FB_MotionStage, etc., for this function block to work properly.

    PMPS handling is done via database lookups by setting sPmpsState on each position state and on
    the transition state input appropriately.
*)
VAR_IN_OUT
    // The 1st motor to move
    stMotionStage1: ST_MotionStage;
    // The 2nd motor to move
    stMotionStage2: ST_MotionStage;
    // All possible position states for motor 1, including unused/invalid states.
    {attribute 'pytmc' := '
        pv: STATE:M1
        io: io
        expand: :%.2d
    '}
    astPositionState1: ARRAY[1..GeneralConstants.MAX_STATES] OF ST_PositionState;
    // All possible position states for motor 2, including unused/invalid states.
    {attribute 'pytmc' := '
        pv: STATE:M2
        io: io
        expand: :%.2d
    '}
    astPositionState2: ARRAY[1..GeneralConstants.MAX_STATES] OF ST_PositionState;
    // Set this to a nonzero value to request a new move. It will be reset to zero every cycle. This should be hooked up to a user's EPICS enum input.
    eEnumSet: UINT;
    // The current state index, or zero if we are not at a state. This should be hooked up to a user's EPICS enum output.
    eEnumGet: UINT;
    // The fast fault output to fault to.
    fbFFHWO: FB_HardwareFFOutput;
    // The arbiter to request beam conditions from.
    fbArbiter: FB_Arbiter;
END_VAR
VAR_INPUT
    // Set this to TRUE to enable input state moves, or FALSE to disable them.
    bEnableMotion: BOOL;
    // Set this to TRUE to enable beam parameter checks, or FALSE to disable them.
    bEnableBeamParams: BOOL;
    // Set this to TRUE to enable position limit checks, or FALSE to disable them.
    bEnablePositionLimits: BOOL;
    // The name of the device for use in the PMPS DB lookup and diagnostic screens.
    sDeviceName: STRING;
    // The name of the transition state in the PMPS database.
    sTransitionKey: STRING;
    // Normal EPICS inputs, gathered into a single struct
    {attribute 'pytmc' := 'pv: STATE'}
    // PMPS EPICS inputs, gathered into a single struct
    stEpicsToPlc: ST_StateEpicsToPlc;
    {attribute 'pytmc' := 'pv: STATE'}
    stPMPSEpicsToPlc: ST_StatePMPSEpicsToPlc;
    // Set this to TRUE to re-read the loaded database immediately (useful for debug)
    bReadDBNow: BOOL;
END_VAR
VAR_OUTPUT
    // Normal EPICS outputs, gathered into a single struct
    {attribute 'pytmc' := 'pv: STATE'}
    stPlcToEpics: ST_StatePlcToEpics;
    // PMPS EPICS outputs, gathered into a single struct
    {attribute 'pytmc' := 'pv: STATE'}
    stPMPSPlcToEpics: ST_StatePMPSPlcToEpics;
    // The PMPS database lookup associated with the current position state.
    stDbStateParams: ST_DbStateParams;
END_VAR
VAR
    fbCore: FB_PositionStateND_Core;
    fbPMPSCore: FB_PositionStatePMPSND_Core;
    astMotionStageMax: ARRAY[1..MotionConstants.MAX_STATE_MOTORS] OF ST_MotionStage;
    astPositionStateMax: ARRAY[1..MotionConstants.MAX_STATE_MOTORS] OF ARRAY[1..GeneralConstants.MAX_STATES] OF ST_PositionState;
END_VAR


astMotionStageMax[1] := stMotionStage1;
astMotionStageMax[2] := stMotionStage2;
astPositionStateMax[1] := astPositionState1;
astPositionStateMax[2] := astPositionState2;

fbCore(
    astMotionStageMax:=astMotionStageMax,
    astPositionStateMax:=astPositionStateMax,
    stEpicsToPlc:=stEpicsToPlc,
    stPlcToEpics:=stPlcToEpics,
    eEnumSet:=eEnumSet,
    eEnumGet:=eEnumGet,
    bEnable:=bEnableMotion,
    nActiveMotorCount:=2,
    nCurrGoal=>,
);
fbPMPSCore(
    astMotionStageMax:=astMotionStageMax,
    astPositionStateMax:=astPositionStateMax,
    stEpicsToPlc:=stEpicsToPlc,
    stPMPSEpicsToPlc:=stPMPSEpicsToPlc,
    stPlcToEpics:=stPlcToEpics,
    stPMPSPlcToEpics:=stPMPSPlcToEpics,
    fbFFHWO:=fbFFHWO,
    fbArbiter:=fbArbiter,
    bEnableBeamParams:=bEnableBeamParams,
    bEnablePositionLimits:=bEnablePositionLimits,
    nActiveMotorCount:=2,
    sDeviceName:=sDeviceName,
    sTransitionKey:=sTransitionKey,
    nCurrGoal:=fbCore.nCurrGoal,
    bReadDBNow:=bReadDBNow,
    stDbStateParams=>stDbStateParams,
);

stMotionStage1 := astMotionStageMax[1];
stMotionStage2 := astMotionStageMax[2];
astPositionState1 := astPositionStateMax[1];
astPositionState2 := astPositionStateMax[2];

END_FUNCTION_BLOCK

// POUs/Motion/PMPS/FB_MotionReadPMPSDBND
FUNCTION_BLOCK FB_MotionReadPMPSDBND
(*
    When we read the JSON PMPS database file, update the lookup parameters for one state mover.
    It is a building block not meant for use outside of lcls-twincat-motion.

    This is intended to support one N-dimensional state motion function block.
    The keys for the database lookup can be set on any of the motor's position states.
    Each of them have an allocated state.stPMPS.sPmpsState STRING parameter.
    If there is a conflict and two of the motors disagree on parameter lookups, that will
    be a fast fault.

    When the global JSON read function block is no longer busy and has no errors,
    we will assume that the file has been read and we will update the parameters here.

    This will also re-read in the event that the input position state keys change in any way,
    provided that we've read once before.
*)
VAR_IN_OUT
    // Each motor's respective position states along its direction. These will not be modified.
    astPositionState: ARRAY[1..MotionConstants.MAX_STATE_MOTORS] OF ARRAY[1..GeneralConstants.MAX_STATES] OF ST_PositionState;
    // Hardware output to fault to if there is a problem.
    fbFFHWO: FB_HardwareFFOutput;
END_VAR
VAR_INPUT
    // The database lookup key for the transition state. This has no corresponding ST_PositionState.
    sTransitionKey: STRING;
    // A name to use for fast faults, etc.
    sDeviceName: STRING;
    // For debug: set this to TRUE in online mode to read the database immediately.
    bReadNow: BOOL;
END_VAR
VAR_OUTPUT
    // The raw lookup results from this FB. Index 0 is the transition beam, the rest of the indices match the state positions.
    astDbStateParams: ARRAY[0..GeneralConstants.MAX_STATES] OF ST_DbStateParams;
    // TRUE if we've had at least one successful read.
    bFirstReadDone: BOOL;
    // This will be set to TRUE if there was an error reading from the database.
    bError: BOOL;
END_VAR
VAR
    ffError: FB_FastFault;
    fbReadPmpsDb: FB_JsonDocToSafeBP;
    ftDbBusy: F_TRIG;
    ftRead: F_TRIG;
    bReadPmpsDb: BOOL;
    nIterMotor: DINT;
    nIterState: DINT;
    nIterState2: DINT;
    sLoopNewKey: STRING;
    sLoopPrevKey: STRING;
    abStateError: ARRAY[0..GeneralConstants.MAX_STATES] OF BOOL;
    asLookupKeys: ARRAY[0..GeneralConstants.MAX_STATES] OF STRING;
    asPrevLookupKeys: ARRAY[0..GeneralConstants.MAX_STATES] OF STRING;
    bNewKeys: BOOL;
    sTempBackfill: STRING;
END_VAR


SelectLookupKeys();
ReadDatabase();
RunFastFaults();
BackfillInfo();

ACTION BackfillInfo:

// Put the results of the PMPS lookup back to the motion states
// This is purely for debugging purposes, as only the astDbStateParams output is used by the libraries.

// Copy everything except for the lookup key: avoid clobbering the user's original keys
// Do it this way instead of one element at a time to be forwards-compatible with any future additions to the db struct
FOR nIterState := 1 TO GeneralConstants.MAX_STATES DO
    FOR nIterMotor := 1 TO MotionConstants.MAX_STATE_MOTORS DO
        sTempBackfill := astPositionState[nIterMotor][nIterState].stPMPS.sPmpsState;
        astPositionState[nIterMotor][nIterState].stPMPS := astDbStateParams[nIterState];
        astPositionState[nIterMotor][nIterState].stPMPS.sPmpsState := sTempBackfill;
    END_FOR
END_FOR
END_ACTION

ACTION ReadDatabase:

// Read the database at the right timing
ftDbBusy(CLK:=MOTION_GVL.fbPmpsFileReader.bBusy);
IF ftDbBusy.Q THEN
    bReadPmpsDb S= NOT MOTION_GVL.fbPmpsFileReader.bError;
END_IF

bReadPmpsDb S= bFirstReadDone AND bNewKeys;
bReadPmpsDb S= bReadNow;
bReadNow := FALSE;

fbReadPmpsDb(
    bExecute:=bReadPmpsDb,
    jsonDoc:=PMPS_GVL.BP_jsonDoc,
    sDeviceName:=sDeviceName,
    io_fbFFHWO:=fbFFHWO,
    arrStates:=astDbStateParams,
);
bReadPmpsDb R= NOT fbReadPmpsDb.bBusy;

ftRead(CLK:=fbReadPmpsDb.bBusy);
bFirstReadDone S= ftRead.Q AND NOT fbReadPmpsDb.bError;
END_ACTION

ACTION RunFastFaults:

ffError(
    i_xOK:=NOT bError,
    i_xAutoReset:=TRUE,
    i_DevName:=sDeviceName,
    i_Desc:='Programmer error selecting state names in ND motion FB',
    i_TypeCode:=E_MotionFFType.INTERNAL_ERROR,
    io_fbFFHWO:=fbFFHWO,
);
END_ACTION

ACTION SelectLookupKeys:

// Fill the lookup key information in astDbStateParams based on the strings from astPositionState and sTransitionKey.

// Start by emptying any pre-existing values
FOR nIterState := 0 TO GeneralConstants.MAX_STATES DO
    asLookupKeys[nIterState] := '';
    abStateError[nIterState] := FALSE;
END_FOR

// Transition key is simple
asLookupKeys[0] := sTransitionKey;

// The other keys might be at different points in the astPositionState array.
// Try all of the posibilities, set error if we end up overwriting something.

// Outer loop: index of each motor at this position state
FOR nIterMotor := 1 TO MotionConstants.MAX_STATE_MOTORS DO
    // Inner loop: index of each position state for this motor
    FOR nIterState := 1 TO GeneralConstants.MAX_STATES DO
        sLoopNewKey := astPositionState[nIterMotor][nIterState].stPMPS.sPmpsState;
        IF sLoopNewKey <> '' THEN
            // We have a new key, start doing things
            sLoopPrevKey := asLookupKeys[nIterState];
            IF sLoopPrevKey = '' OR sLoopPrevKey = sLoopNewKey THEN
                // No key yet, or exactly the same key (redudant programmer)
                asLookupKeys[nIterState] := sLoopNewKey;
            ELSE
                // We already had a different key! Don't just override it, have an error!
                bError := TRUE;
                abStateError[nIterState] := TRUE;
            END_IF
        END_IF
    END_FOR
END_FOR

// Check for duplicated sPmpsState strings
FOR nIterState := 0 TO GeneralConstants.MAX_STATES DO
    FOR nIterState2 := 0 TO nIterState DO
        IF nIterState <> nIterState2 THEN
            IF asLookupKeys[nIterState] = asLookupKeys[nIterState2] THEN
                // Duplicated key, we need an error and a flag in both spots
                bError := TRUE;
                abStateError[nIterState] := TRUE;
                abStateError[nIterState2] := TRUE;
            END_IF
        END_IF
    END_FOR
END_FOR

// Clear the erroneous states so they won't be used as lookups
IF bError THEN
    FOR nIterState := 0 TO GeneralConstants.MAX_STATES DO
        IF abStateError[nIterState] THEN
            asLookupKeys[nIterState] := '';
        END_IF
    END_FOR
END_IF

// Copy the keys into the db state params
FOR nIterState := 0 TO GeneralConstants.MAX_STATES DO
    astDbStateParams[nIterState].sPmpsState := asLookupKeys[nIterState];
END_FOR

// Check if the keys changed from prev cycle
bNewKeys := FALSE;
FOR nIterState := 0 TO GeneralConstants.MAX_STATES DO
    IF asLookupKeys[nIterState] <> asPrevLookupKeys[nIterState] THEN
        bNewKeys := TRUE;
        EXIT;
    END_IF
END_FOR

// Save prev keys for next cycle
asPrevLookupKeys := asLookupKeys;
END_ACTION

END_FUNCTION_BLOCK

// POUs/Motion/PMPS/FB_MotionBPTM

FUNCTION_BLOCK FB_MotionBPTM
(*
    This function block handles the beam parameter transition manager for a group of motors moving together to a destination with shared beam state.
    stGoalParams and stTransParams are required arguments and must not share IDs with other state parameters in the PLC.

    This is a building block not intended for use outside of lcls-twincat-motion.
*)
VAR_IN_OUT
    // Array of motors that will move for this beam transition
    astMotionStage: ARRAY[1..MotionConstants.MAX_STATE_MOTORS] OF ST_MotionStage;
    // The arbiter to request beam states from
    fbArbiter: FB_Arbiter;
    // The fast fault output to fault to
    fbFFHWO: FB_HardwareFFOutput;
    // The parameters we want to transition to
    stGoalParams: ST_DbStateParams;
    // The parameters we want to use during the transition
    stTransParams: ST_DbStateParams;
END_VAR
VAR_INPUT
    // The number of motors we're actually using
    nActiveMotorCount: UINT;
    // Set to TRUE to use the BPTM, FALSE to stop using the BPTM.
    bEnable: BOOL;
    // TRUE if we're at the physical state that matches the goal parameters
    bAtState: BOOL;
    // A device name to use in the GUI
    sDeviceName: STRING;
    // How long to wait for parameters before timing out
    tArbiterTimeout: TIME := T#1s;
    // Whether to fault and move on timeout (TRUE) or to wait (FALSE)
    bMoveOnArbiterTimeout: BOOL := TRUE;
    // Set to TRUE when it is safe to reset the BPTM timeout fast fault, to reset it early.
    bResetBPTMTimeout: BOOL;
END_VAR
VAR_OUTPUT
    // This becomes TRUE when the motors are allowed to move to their destinations.
    bTransitionAuthorized: BOOL;
    // This becomes TRUE once the full beam transition is done.
    bDone: BOOL;
    // TRUE if we're using a bad motor count
    bMotorCountError: BOOL;
END_VAR
VAR
    bptm: BeamParameterTransitionManager;
    bDoneMoving: BOOL;
    nPrevID: UDINT;
    nIndex: DINT;

    bInternalAuth: BOOL;
    bDoneResetQueued: BOOL;

    tonArbiter: TON;
    bArbiterTimeout: BOOL;
    ffBPTMTimeoutAndMove: FB_FastFault;
    ffBPTMError: FB_FastFault;
END_VAR


CheckCount();
IF NOT bMotorCountError THEN
    SetDoneMoving();
    IF bEnable THEN
        RunBPTM();
        HandleTimeout();
    END_IF
END_IF

ACTION CheckCount:

// Make sure the motor count is valid (positive, nonzero, less or equal to the max)
bMotorCountError S= nActiveMotorCount <= 0;
bMotorCountError S= nActiveMotorCount > MotionConstants.MAX_STATE_MOTORS;
END_ACTION

ACTION HandleTimeout:

// Measure the time that the bptm is busy
tonArbiter(
    IN:=bptm.bBusy,
    PT:=tArbiterTimeout,
    Q=>bArbiterTimeout,
);
bTransitionAuthorized := bInternalAuth OR (bArbiterTimeout AND bMoveOnArbiterTimeout);

// Trip the beam for BPTM timeouts if we want to move
// Only reset at safe beam OR at no bptm errors (some other FF should catch additional issues)
ffBPTMTimeoutAndMove.i_xOK := NOT (bArbiterTimeout AND bMoveOnArbiterTimeout);
ffBPTMTimeoutAndMove.i_xReset S= bResetBPTMTimeout OR (bptm.bDone AND NOT bptm.bError);
ffBPTMTimeoutAndMove(
    i_DevName := sDeviceName,
    i_Desc := 'BPTM Timeout',
    i_TypeCode := E_MotionFFType.BPTM_TIMEOUT,
    io_fbFFHWO := fbFFHWO,
);
END_ACTION

ACTION RunBPTM:

bptm(
    fbArbiter:=fbArbiter,
    i_sDeviceName:=sDeviceName,
    i_TransitionAssertionID:=stTransParams.nRequestAssertionID,
    i_stTransitionAssertion:=stTransParams.stBeamParams,
    i_nRequestedAssertionID:=stGoalParams.nRequestAssertionID,
    i_stRequestedAssertion:=stGoalParams.stBeamParams,
    i_xDoneMoving:=bDoneMoving AND bAtState,
    stCurrentBeamParameters:=PMPS_GVL.stCurrentBeamParameters,
    q_xTransitionAuthorized=>bInternalAuth,
    bDone=>bDone,
);

// Trip the beam for BPTM Errors
ffBPTMError.i_xOK := NOT bptm.bError;
ffBPTMError.i_xReset S= bptm.bDone AND NOT bptm.bError;
ffBPTMError(
    i_DevName := sDeviceName,
    i_Desc := 'BPTM error, state transition failed',
    i_TypeCode := E_MotionFFType.BPTM_ERROR,
    io_fbFFHWO := fbFFHWO,
);
END_ACTION

ACTION SetDoneMoving:

// Set bDoneMoving if all the motors are done
bDoneMoving := TRUE;
FOR nIndex := 1 TO nActiveMotorCount DO
    bDoneMoving := bDoneMoving AND NOT astMotionStage[nIndex].bBusy AND NOT astMotionStage[nIndex].bExecute;
END_FOR
// Reset bDoneMoving if the goal has changed to reset bptm's motor done for an in-place transition
// This allows us to change to a new beam state without requiring a motor state change
// BPTM only checks for this "done" transition after the transition has been authorized, so we may need to wait
bDoneResetQueued S= nPrevID <> stGoalParams.nRequestAssertionID;
bDoneMoving R= bDoneResetQueued AND bptm.q_xTransitionAuthorized;
bDoneResetQueued R= bptm.q_xTransitionAuthorized;
nPrevID := stGoalParams.nRequestAssertionID;
END_ACTION

END_FUNCTION_BLOCK

// POUs/Motion/PMPS/FB_MotionClearAsserts
FUNCTION_BLOCK FB_MotionClearAsserts
(*
    Clear all of the PMPS asserts related to a states mover.
*)
VAR_IN_OUT
    // All states to deactivate: transition + the static position states
    astDbStateParams: ARRAY[0..GeneralConstants.MAX_STATES] OF ST_DbStateParams;
    // The arbiter who made the PMPS assert requests
    fbArbiter: FB_ARBITER;
END_VAR
VAR_INPUT
    // Clear asserts on rising edge
    bExecute: BOOL;
END_VAR
VAR_OUTPUT
END_VAR
VAR
    rtExec: R_TRIG;
    nIter: DINT;
END_VAR


rtExec(CLK:=bExecute);
IF rtExec.Q THEN
    FOR nIter := 0 TO GeneralConstants.MAX_STATES DO
        fbArbiter.RemoveRequest(astDbStateParams[nIter].nRequestAssertionID);
    END_FOR
END_IF

END_FUNCTION_BLOCK

// POUs/Motion/PMPS/FB_StatePMPSEnablesND
FUNCTION_BLOCK FB_StatePMPSEnablesND
(*
    Function block to set virtual limit enables using MC_POWER for multidimensional state movers.
    It is a building block not meant for use outside of lcls-twintcat-motion.

    Each motor has a virtual "allowed" range of motion based on its goal position.
    Motors can move toward their goal delta ranges or within them, but not away from these ranges.
*)
VAR_IN_OUT
    // The motors with a combined N-dimensional state
    astMotionStage: ARRAY[1..MotionConstants.MAX_STATE_MOTORS] OF ST_MotionStage;
    // Each motor's respective position states along its direction
    astPositionState: ARRAY[1..MotionConstants.MAX_STATE_MOTORS] OF ARRAY[1..GeneralConstants.MAX_STATES] OF ST_PositionState;
    // Hardware output to fault to if there is a problem.
    fbFFHWO: FB_HardwareFFOutput;
END_VAR
VAR_INPUT
    // Whether or not to do anything
    bEnable: BOOL;
    // The number of motors we're actually using
    nActiveMotorCount: UINT;
    // The state that the motors are moving to, along dimension 2 of the position state array. This may be the same as the current state.
    nGoalStateIndex: UINT;
    // A name to use for this state mover in the case of fast faults.
    sDeviceName: STRING;
    // Set to TRUE to put motors into maintenance mode. This allows us to freely move the motors at the cost of a fast fault.
    bMaintMode: BOOL;
    // The overal PMPS FB state
    eStatePMPSStatus: E_StatePMPSStatus;
    // Connect from bptm bTransitionAuthorized
    bTransitionAuthorized: BOOL;
END_VAR
VAR_OUTPUT
    // Per-motor enable state we send to MC_Power. This is a pass-through from stMotionStage.
    abEnabled: ARRAY[1..MotionConstants.MAX_STATE_MOTORS] OF BOOL;
    // Per-motor forward enable state we send to MC_Power. This may be a pass-through or an override to FALSE.
    abForwardEnabled: ARRAY[1..MotionConstants.MAX_STATE_MOTORS] OF BOOL;
    // Per-motor backwards enable state we send to MC_Power. This may be a pass-through or an override to FALSE.
    abBackwardEnabled: ARRAY[1..MotionConstants.MAX_STATE_MOTORS] OF BOOL;
    // Per-motor TRUE if there is a valid goal position and FALSE otherwise. This makes a fast fault if FALSE.
    abValidGoal: ARRAY[1..MotionConstants.MAX_STATE_MOTORS] OF BOOL;
    // Set to TRUE if the arrays have mismatched sizing. For this FB, this means the motor won't ever get an enable.
    bMotorCountError: BOOL;
END_VAR
VAR
    // The individual state limit function blocks
    afbStateEnables: ARRAY[1..MotionConstants.MAX_STATE_MOTORS] OF FB_StatePMPSEnables;
    ffMaint: FB_FastFault;
    ffProgrammerError: FB_FastFault;
    nIter: DINT;
END_VAR


CheckCount();
IF NOT bMotorCountError THEN
    DoLimits();
END_IF
RunFastFaults();

ACTION CheckCount:

// Make sure the motor count is valid (positive, nonzero, less or equal to the max)
bMotorCountError S= nActiveMotorCount <= 0;
bMotorCountError S= nActiveMotorCount > MotionConstants.MAX_STATE_MOTORS;
END_ACTION

ACTION DoLimits:

FOR nIter := 1 TO nActiveMotorCount DO
    afbStateEnables[nIter](
        stMotionStage:=astMotionStage[nIter],
        astPositionState:=astPositionState[nIter],
        fbFFHWO:=fbFFHWO,
        bEnable:=bEnable AND NOT bMaintMode,
        nGoalStateIndex:=nGoalStateIndex,
        eStatePMPSStatus:=eStatePMPSStatus,
        bTransitionAuthorized:=bTransitionAuthorized,
        bEnabled=>abEnabled[nIter],
        bForwardEnabled=>abForwardEnabled[nIter],
        bBackwardEnabled=>abBackwardEnabled[nIter],
        bValidGoal=>abValidGoal[nIter],
    );
END_FOR
END_ACTION

ACTION RunFastFaults:

ffMaint(
    i_xOK := NOT bMaintMode,
    i_xAutoReset := TRUE,
    i_DevName := sDeviceName,
    i_Desc := 'Device is in maintenance mode',
    i_TypeCode := E_MotionFFType.MAINT_MODE,
    io_fbFFHWO := fbFFHWO,
);

ffProgrammerError(
    i_xOK:=NOT bMotorCountError,
    i_xAutoReset:=TRUE,
    i_DevName:=sDeviceName,
    i_Desc:='Programmer error picking motor count',
    i_TypeCode:=E_MotionFFType.INTERNAL_ERROR,
    io_fbFFHWO:=fbFFHWO,
);
END_ACTION

END_FUNCTION_BLOCK

// POUs/Motion/PMPS/FB_StatePMPSEnables
FUNCTION_BLOCK FB_StatePMPSEnables
(*
    Function block to set virtual limit enables using MC_POWER for single dimensional state movers.
    It is a building block not meant for use outside of lcls-twintcat-motion.

    Each motor has a virtual "allowed" range of motion based on its goal position.
    When not at the goal, the motor can only move toward the goal.
    When at the goal, the motor can move within the position's delta.

    With no goals or other strange states, the motor is permitted to move in either direction
    to help restore it to a known position.
*)
VAR_IN_OUT
    // The motor with a position state.
    stMotionStage: ST_MotionStage;
    // All possible position states for this motor.
    astPositionState: ARRAY[1..GeneralConstants.MAX_STATES] OF ST_PositionState;
    // Hardware output to fault to if there is a problem.
    fbFFHWO: FB_HardwareFFOutput;
END_VAR
VAR_INPUT
    // If TRUE, do the limits as normal. If FALSE, allow all moves regardless of the limits defined here.
    bEnable: BOOL;
    // The state that the motor is moving to.
    nGoalStateIndex: UINT;
    // The overal PMPS FB state
    eStatePMPSStatus: E_StatePMPSStatus;
    // Connect to the BPTM
    bTransitionAuthorized: BOOL;
END_VAR
VAR_OUTPUT
    // The enable state we send to MC_Power. This is a pass-through from stMotionStage.
    bEnabled: BOOL;
    // The forward enable state we send to MC_Power. This may be a pass-through or an override to FALSE.
    bForwardEnabled: BOOL;
    // The backwards enable state we send to MC_Power. This may be a pass-through or an override to FALSE.
    bBackwardEnabled: BOOL;
    // TRUE if there is a valid goal position and FALSE otherwise. This makes a fast fault if FALSE.
    bValidGoal: BOOL;
END_VAR
VAR
    mc_power: MC_POWER;
    nPrevStateIndex: DINT;
    fLowerPos: LREAL;
    fUpperPos: LREAL;
    ffNoGoal: FB_FastFault;
END_VAR


GetBounds();
SetEnables();
ApplyEnables();
RunFastFaults();

ACTION ApplyEnables:

(*
    This action takes runs MC_POWER appropriately
    given the motor's own enables and the results of this FB's checks.
*)
bEnabled := stMotionStage.bAllEnable;
bForwardEnabled := bForwardEnabled AND stMotionStage.bAllForwardEnable;
bBackwardEnabled := bBackwardEnabled AND stMotionStage.bAllBackwardEnable;

CASE eStatePMPSStatus OF
    E_StatePMPSStatus.UNKNOWN:
        stMotionStage.bSafetyReady := FALSE;
    E_StatePMPSStatus.TRANSITION:
        stMotionStage.bSafetyReady := bTransitionAuthorized;
        bForwardEnabled R= NOT bTransitionAuthorized;
        bBackwardEnabled R= NOT bTransitionAuthorized;
    E_StatePMPSStatus.AT_STATE:
        stMotionStage.bSafetyReady := stMotionStage.bExecute;
    E_StatePMPSStatus.DISABLED:
        stMotionStage.bSafetyReady := TRUE;
END_CASE

mc_power(
    Axis:=stMotionStage.Axis,
    Enable:=bEnabled,
    Enable_Positive:=bForwardEnabled,
    Enable_Negative:=bBackwardEnabled,
);
END_ACTION

ACTION GetBounds:

(*
    This action sets fLowerPos and fUpperPos based on our goal position.
*)
IF nGoalStateIndex > 0 AND nGoalStateIndex <= GeneralConstants.MAX_STATES THEN
    IF astPositionState[nGoalStateIndex].bValid AND astPositionState[nGoalStateIndex].bUpdated THEN
        bValidGoal := TRUE;
        fLowerPos := astPositionState[nGoalStateIndex].fPosition - ABS(astPositionState[nGoalStateIndex].fDelta);
        fUpperPos := astPositionState[nGoalStateIndex].fPosition + ABS(astPositionState[nGoalStateIndex].fDelta);
    ELSE
        bValidGoal := FALSE;
    END_IF
ELSE
    bValidGoal := FALSE;
END_IF
END_ACTION

ACTION RunFastFaults:

ffNoGoal(
    i_xOK:=bValidGoal,
    i_xAutoReset:=TRUE,
    i_DevName:=stMotionStage.sName,
    i_Desc:='Invalid goal position in state move',
    i_TypeCode:=E_MotionFFType.INVALID_GOAL,
    io_fbFFHWO:=fbFFHWO,
);
END_ACTION

ACTION SetEnables:

(*
    This action sets bForwardEnable and bBackwardEnable based on
    the current position and the calculated bounds.
*)
IF bValidGoal AND bEnable THEN
    bForwardEnabled := stMotionStage.stAxisStatus.fActPosition < fUpperPos;
    bBackwardEnabled := stMotionStage.stAxisStatus.fActPosition > fLowerPos;
ELSE
    // Either invalid state with a fault or FB not enabled
    bForwardEnabled := TRUE;
    bBackwardEnabled := TRUE;
END_IF
END_ACTION

END_FUNCTION_BLOCK

// POUs/Motion/PMPS/FB_MiscStatesErrorFFO
FUNCTION_BLOCK FB_MiscStatesErrorFFO
(*
    A catch-all for miscellaneous state FFOs that are not better organized elsewhere.
    Contains the following fast faults:
    - ffBeamParamsOK: trip the beam if the beam parameters are not safe enough for our current (known) state
    - ffZeroRate: trip the beam if we've asked for zero rate (as a shortcut)
    - ffUnknown: trip the beam if we're at an unknown state and our transition id is not asserted.
    - ffDebounce: trip the beam (no autoreset) if ffBeamParamsOK fast faults fault on and off multiple times too quickly.
      This solves an issue where ffBeamParamsOK might solve its own problem and creating a blinking fast fault issue.

    The inputs are mostly outputs of non-pmps function blocks and heavily-reused info like state details.
*)
VAR_IN_OUT
    // The arbiter to request beam states from
    fbArbiter: FB_Arbiter;
    // The fast fault output to fault to
    fbFFHWO: FB_HardwareFFOutput;
END_VAR
VAR_INPUT
    // A name to link to these fast faults
    sDeviceName: STRING;
    // Current requested beam details: either a known state or the transition beam
    stCurrentBeamReq: ST_BeamParams;
    // TRUE if we're at a known state (doesn't matter which)
    bKnownState: BOOL;
    // Lookup ID of the transition beam
    nTransitionID: DWORD;
END_VAR
VAR_OUTPUT
END_VAR
VAR CONSTANT
    // Number of consecutive trips before we debounce
    nMaxTrips: UINT := 5;
    // Decrease trip count by 1 after this much time has passed
    tTripReset: TIME := T#1s;
END_VAR
VAR
    // If the beam parameters are wrong, it is a fault! This encompasses all unknown arbiter-related errors.
    ffBeamParamsOk: FB_FastFault;
    // If we asked for zero rate (NC or SC) then we can cut the beam early. This is somewhat redundant.
    ffZeroRate: FB_FastFault;
    // Trip the beam for unknown state
    ffUnknown: FB_FastFault;
    // Trip the beam (no autoreset) if ffBeamParamsOK faults/resets multiple times too quickly.
    ffDebounce: FB_FastFault;

    // Number of consecutive trips so far
    nTripCount: UINT;
    // Increase by 1 whenever there is a fault (rising edge)
    ftTripCount: F_TRIG;
    // Decrease trip count by 1 each timeout
    tonTripCount: TON;
    // TRUE on only the first cycle
    bFirstCycle: BOOL := TRUE;
END_VAR


ffBeamParamsOk(
    i_xOK:=F_SafeBPCompare(PMPS_GVL.stCurrentBeamParameters, stCurrentBeamReq),
    i_xAutoReset:=TRUE,
    i_DevName:=sDeviceName,
    i_Desc:='Beam parameter mismatch',
    i_TypeCode:=E_MotionFFType.BP_MISMATCH,
    io_fbFFHWO:=fbFFHWO);

CASE PMPS_GVL.stCurrentBeamParameters.nMachineMode OF
    // NC mode
    1: ffZeroRate.i_xOK := stCurrentBeamReq.nRate > 0;
    // SC mode
    2: ffZeroRate.i_xOK := stCurrentBeamReq.nBCRange > 0;
ELSE
    // Ambiguous or new mode
    ffZeroRate.i_xOK := stCurrentBeamReq.nRate > 0 AND stCurrentBeamReq.nBCRange > 0;
END_CASE

ffZeroRate(
    i_xAutoReset := TRUE,
    i_DevName := sDeviceName,
    i_Desc := 'Device requesting zero rate',
    i_TypeCode := E_MotionFFType.ZERO_RATE,
    io_fbFFHWO := fbFFHWO,
);

ffUnknown(
    i_xOK := bknownState OR fbArbiter.CheckRequestInPool(nReqID:=nTransitionID),
    i_xAutoReset := TRUE,
    i_DevName := sDeviceName,
    i_Desc := 'Unknown position between moves',
    i_TypeCode := E_MotionFFType.NOT_A_STATE,
    io_fbFFHWO := fbFFHWO,
);

ftTripCount(CLK:=ffBeamParamsOk.i_xOK);

IF ftTripCount.Q THEN
    nTripCount := nTripCount + 1;
END_IF

tonTripCount(
    IN:=NOT tonTripCount.Q,
    PT:=tTripReset,
);
IF tonTripCount.Q AND nTripCount > 0 THEN
    nTripCount := nTripCount - 1;
END_IF

// This is required for non-autoresetting FBs to come up in a beam permitted state
ffDebounce.i_xReset S= bFirstCycle;
ffDebounce(
    i_xOK := nTripCount < 5,
    i_xAutoReset := FALSE,
    i_DevName := sDeviceName,
    i_Desc := 'Tripped beam parameter mismatch off/on too many times, hold off',
    i_TypeCode := E_MotionFFType.TOO_MANY_TRIPS,
    io_fbFFHWO := fbFFHWO,
);
ffDebounce.i_xReset R= bFirstCycle;
bFirstCycle := FALSE;

END_FUNCTION_BLOCK

// POUs/Motion/PMPS/FB_PerMotorFFOND
FUNCTION_BLOCK FB_PerMotorFFOND
(*
    PMPS fast faults that must be done per motor, rather than per state, based purely
    on the motor status and not other PMPS considerations.

    These currently include:
    - Fault if the encoder has an error. Every other protection is based on the encoder,
      so we can't trust anything if the encoder is faulting.
*)
VAR_IN_OUT
    // All motors associated with the state mover.
    astMotionStage: ARRAY[1..MotionConstants.MAX_STATE_MOTORS] OF ST_MotionStage;
    // Fast fault output to fault to.
    fbFFHWO: FB_HardwareFFOutput;
END_VAR
VAR_INPUT
    // The number of motors we're actually using
    nActiveMotorCount: UINT;
    // Identifying name to use in group fast faults
    sDeviceName: STRING;
END_VAR
VAR_OUTPUT
    // Set to TRUE if the arrays don't have the same bounds. In this FB, that's an automatic fault.
    bMotorCountError: BOOL;
END_VAR
VAR
    afbEncError: ARRAY[1..MotionConstants.MAX_STATE_MOTORS] OF FB_EncErrorFFO;
    ffProgrammerError: FB_FastFault;
    nIter: DINT;
END_VAR


CheckCount();
IF NOT bMotorCountError THEN
    HandleLoops();
END_IF
HandleFFO();

ACTION CheckCount:

// Make sure the motor count is valid (positive, nonzero, less or equal to the max)
bMotorCountError S= nActiveMotorCount <= 0;
bMotorCountError S= nActiveMotorCount > MotionConstants.MAX_STATE_MOTORS;
END_ACTION

ACTION HandleFFO:

ffProgrammerError(
    i_xOK:=NOT bMotorCountError,
    i_xAutoReset:=TRUE,
    i_DevName:=sDeviceName,
    i_Desc:='Programmer error picking motor count',
    i_TypeCode:=E_MotionFFType.INTERNAL_ERROR,
    io_fbFFHWO:=fbFFHWO,
);
END_ACTION

ACTION HandleLoops:

FOR nIter := 1 TO nActiveMotorCount DO
    afbEncError[nIter](
        stMotionstage:=astMotionStage[nIter],
        fbFFHWO:=fbFFHWO,
        bAutoReset:=TRUE,
    );
END_FOR
END_ACTION

END_FUNCTION_BLOCK

// POUs/Motion/PMPS/FB_EncErrorFFO
FUNCTION_BLOCK FB_EncErrorFFO
(*
    Example usage of FB_NCErrorFFO that only counts encoder errors as faults.
*)
VAR_IN_OUT
    // Motion stage to monitor
    stMotionStage: ST_MotionStage;
    // FFO to trip
    fbFFHWO: FB_HardwareFFOutput;
END_VAR
VAR_INPUT
    // Reset the fault
    bReset: BOOL;
    // Auto reset the fault
    bAutoReset: BOOL;
END_VAR
VAR_OUTPUT
    // Quick way for nearby code to check if this block has tripped the FFO.
    bTripped: BOOL;
END_VAR
VAR
    fbNCErrorFFO: FB_NCErrorFFO := (
        nLowErrorId := 16#4400,
        nHighErrorId := 16#44FF,
        sDesc := 'Encoder error');
END_VAR

fbNCErrorFFO(
    stMotionStage := stMotionStage,
    fbFFHWO := fbFFHWO,
    bReset := bReset,
    bAutoReset := bAutoReset,
    bTripped => bTripped);

END_FUNCTION_BLOCK

// POUs/Motion/PMPS/FB_NCErrorFFO
FUNCTION_BLOCK FB_NCErrorFFO
(*
    Configure a ST_MotionStage to trigger an FFO when we have an error.

    This can be configured to only apply to specific error ranges,
    though the default is the normal 16#4XXX NC error range. The error
    ranges are:
    16#40XX General Errors
    16#41XX Channel Errors
    16#42XX Group Errors
    16#43XX Axis Errors
    16#44XX Encoder Errors
    16#45XX Controller Errors
    16#46XX Drive Errors
    16#4AXX Table Errors
    16#4BXX NC PLC Errors
    16#4CXX Kinematic Transformation

    There is also a new extended NC error range, but it is sparsely populated.
    This range is 16#8XXX:
    16#8100 - 16#811F: Bode plot (diagnosis)
    16#8120 - 16#8FFF: Further errors

    To configure multiple ranges, simply use multiple instances of this
    function block.
*)
VAR_IN_OUT
    // Motion stage to monitor
    stMotionStage: ST_MotionStage;
    // FFO to trip
    fbFFHWO: FB_HardwareFFOutput;
END_VAR
VAR_INPUT
    // Reset the fault
    bReset: BOOL;
    // Auto-reset the fault
    bAutoReset: BOOL;
    // The lowest error code that will trip the FFO
    nLowErrorId: UDINT := 16#4000;
    // The highest error code that will trip the FFO
    nHighErrorId: UDINT := 16#4FFF;
    // A description of the fault
    sDesc: STRING := 'Motor error';
END_VAR
VAR_OUTPUT
    // Quick way for nearby code to check if this block has tripped the FFO.
    bTripped: BOOL;
    // Error code sent to PMPS. Is always 16#20XX, where XX is the first two hex in the NC error.
    nErrorTypeCode: UINT;
END_VAR
VAR
    bInit: BOOL;
    stBeamParams: ST_BeamParams;
    fbFF: FB_FastFault;
    rtTrip: R_TRIG;
END_VAR

IF NOT bInit THEN
    fbFF.i_Desc := sDesc;
    IF LEN(stMotionStage.sName) > 0 THEN
        fbFF.i_DevName := stMotionStage.sName;
    ELSE
        fbFF.i_DevName := 'Unnamed Motor';
    END_IF
    bInit := TRUE;
END_IF

bTripped := stMotionStage.bError AND stMotionStage.nErrorId >= nLowErrorId AND stMotionStage.nErrorId <= nHighErrorId;
rtTrip(CLK:=bTripped);
IF rtTrip.Q THEN
    nErrorTypeCode := E_MotionFFType.LOW_RESERVED_NC + UDINT_TO_UINT(SHR(stMotionStage.nErrorId, 8));
    nErrorTypeCode := MIN(nErrorTypeCode, E_MotionFFType.HIGH_RESERVED_NC);
END_IF
fbFF(i_xOK := NOT bTripped,
     i_xReset := bReset,
     i_xAutoReset := bAutoReset,
     i_TypeCode:= nErrorTypeCode,
     io_fbFFHWO := fbFFHWO);

END_FUNCTION_BLOCK

// POUs/Motion/States/FB_StatesInputHandler
FUNCTION_BLOCK FB_StatesInputHandler
(*
    Handle the state enum EPICS input for any of the ND state function blocks.

    The desired behavior is:
    - Trigger a move to a new state when the enum PV is written to
    - Interrupt an ongoing move with a new one if the enum changes mid-move
    - Stop the move if the enum is set to an invalid value
*)
VAR_IN_OUT
    // The user's inputs from EPICS. This is an IN_OUT variable because we will write values back to this to help us detect when the same value is re-caput
    stUserInput: ST_StateEpicsToPlc;
END_VAR
VAR_INPUT
    // The bBusy boolean from the motion FB
    bMoveBusy: BOOL;
    // The starting state number to seed nCurrGoal with
    nStartingState: UINT;
END_VAR
VAR_OUTPUT
    // The goal index to input to the motion FB. This will be clamped to the range 0..GeneralConstants.MAX_STATES
    nCurrGoal: UINT;
    // The bExecute boolean to input to the motion FB
    bExecMove: BOOL;
    // The bReset boolean to input to the motion FB
    bResetMove: BOOL;
END_VAR
VAR
    nState: UINT;
    bInit: BOOL;
    nQueuedGoal: UINT;
    bNewMove: BOOL;
END_VAR
VAR CONSTANT
    IDLE: UINT := 0;
    GOING: UINT := 1;
    WAIT_STOP: UINT := 2;
END_VAR


IF NOT bInit THEN
    bInit := TRUE;
    stUserInput.nSetValue := 0;
    nCurrGoal := nStartingState;
END_IF

bResetMove := stUserInput.bReset;

IF stUserInput.nSetValue <> 0 THEN
    nQueuedGoal := stUserInput.nSetValue;
    bNewMove := TRUE;
END_IF

CASE nState OF
    IDLE:
        IF bNewMove AND nQueuedGoal > 0 AND nQueuedGoal <= GeneralConstants.MAX_STATES THEN
            // New request, currently idle -> ask for a move
            nCurrGoal := nQueuedGoal;
            bExecMove := TRUE;
            bNewMove := FALSE;
        ELSIF bMoveBusy THEN
            // We're moving but used to be idle -> switch to GOING
            nState := GOING;
        END_IF
    GOING:
        IF bNewMove THEN
            // New request, currently moving -> ask for a stop
            nState := WAIT_STOP;
            bExecMove := FALSE;
        ELSIF NOT bMoveBusy THEN
            nState := IDLE;
            nQueuedGoal := 0;
            bExecMove := FALSE;
        END_IF
    WAIT_STOP:
        IF NOT bMoveBusy THEN
            nState := IDLE;
        END_IF
END_CASE

// Help us detect if there is an EPICS put before the next cycle
stUserInput.nSetValue := 0;
stUserInput.bReset := FALSE;

END_FUNCTION_BLOCK

// POUs/Motion/States/Internals/FB_PositionStateInternalND
FUNCTION_BLOCK FB_PositionStateInternalND
(*
    Given a standard ND state setup, call all the required state management FBs.
*)
VAR_IN_OUT
    // All the motors to apply the standard routines to
    astMotionStage: ARRAY[1..MotionConstants.MAX_STATE_MOTORS] OF ST_MotionStage;
    // Each motor's respective position states along its direction
    astPositionState: ARRAY[1..MotionConstants.MAX_STATE_MOTORS] OF ARRAY[1..GeneralConstants.MAX_STATES] OF ST_PositionState;
END_VAR
VAR
    // The individual instantiated internal FBs. Must have the same bounds as astPositionState.
    afbStateInternal: ARRAY[1..MotionConstants.MAX_STATE_MOTORS] OF ARRAY[1..GeneralConstants.MAX_STATES] OF FB_PositionStateInternal;
    nIterMotors: DINT;
    nIterStates: DINT;
END_VAR


FOR nIterMotors := 1 TO MotionConstants.MAX_STATE_MOTORS DO
    FOR nIterStates := 1 TO GeneralConstants.MAX_STATES DO
        afbStateInternal[nIterMotors][nIterStates](
            stMotionStage:=astMotionStage[nIterMotors],
            stPositionState:=astPositionState[nIterMotors][nIterStates],
        );
    END_FOR
END_FOR

END_FUNCTION_BLOCK

// POUs/Motion/States/Internals/FB_PositionStateInternal
FUNCTION_BLOCK FB_PositionStateInternal
(*
    Routines that must be called on all ST_PositionState

    Currently, this FB:
    - ensures that a position state has both a proper encoder count
      and a proper position in engineering units with both of these quantities matching
    - handles the parameter locking feature, which nominally prevents the user from changing
      details about a locked state via EPICS
*)
VAR_IN_OUT
    stMotionStage: ST_MotionStage;
    stPositionState: ST_PositionState;
END_VAR
VAR_OUTPUT
END_VAR
VAR
    fbEncConverter: FB_RawCountConverter;
    fbLock: FB_PositionStateLock;
END_VAR

// Mark that we've been here
stPositionState.bUpdated := TRUE;

// Update pos state's count or egu position as appropriate
IF stMotionStage.bAxisParamsInit THEN
    fbEncConverter(
        stParameters:=stMotionStage.stAxisParameters,
        nCountCheck:=stPositionState.nEncoderCount,
        fPosCheck:=stPositionState.fPosition);
    IF stPositionState.bUseRawCounts THEN
        stPositionState.fPosition := fbEncConverter.fPosGet;
    ELSE
        stPositionState.nEncoderCount := fbEncConverter.nCountGet;
    END_IF
END_IF

// Handle state parameter locking
fbLock(
    stPositionState:=stPositionState,
    bEnable:=stMotionStage.bAxisParamsInit);

END_FUNCTION_BLOCK

// POUs/Motion/States/Helpers/FB_RawCountConverter
FUNCTION_BLOCK FB_RawCountConverter
(*
    Utility function block for converting raw counts to EGU and back
*)
VAR_INPUT
    // Parameters to check against
    stParameters: ST_AxisParameterSet;
    // Optional count to convert to a real position
    nCountCheck: UDINT;
    // Optional position to convert to encoder counts
    fPosCheck: LREAL;
END_VAR
VAR_OUTPUT
    // If converting position, the number of counts
    nCountGet: UDINT;
    // If converting counts, the position
    fPosGet: LREAL;
    // True during a parameter get/calc
    bBusy: BOOL;
    // True after a successful get/calc
    bDone: BOOL;
    // True if the calculation errored
    bError: BOOL;
END_VAR

IF stParameters.fEncScaleFactorInternal <> 0 THEN
    nCountGet := LREAL_TO_UDINT((fPosCheck - stParameters.fEncOffset) / stParameters.fEncScaleFactorInternal);
    fPosGet := nCountCheck * stParameters.fEncScaleFactorInternal + stParameters.fEncOffset;
END_IF

END_FUNCTION_BLOCK

// POUs/Motion/States/Internals/FB_PositionStateLock
FUNCTION_BLOCK FB_PositionStateLock
(*
    Implements immutability for a locked ST_PositionState
    Once this is called the first time, the parameters at the time of the call will be restored on all subsequent calls.
*)
VAR_IN_OUT
    stPositionState: ST_PositionState;
END_VAR
VAR_INPUT
    bEnable: BOOL;
END_VAR
VAR
    stCachedPositionState: ST_PositionState;
    bInit: BOOL := FALSE;
END_VAR

IF bEnable THEN
    // Force values to be cached if we've cached something
    IF bInit AND stPositionState.bLocked THEN
        stPositionState.sName := stCachedPositionState.sName;
        stPositionState.fPosition := stCachedPositionState.fPosition;
        stPositionState.fDelta := stCachedPositionState.fDelta;
        stPositionState.fVelocity := stCachedPositionState.fVelocity;
        stPositionState.fAccel := stCachedPositionState.fAccel;
        stPositionState.fDecel := stCachedPositionState.fDecel;
    // If we haven't cached and we should, make the cache. Note that we skip bLocked, bValid, and bMoveOk
    ELSIF NOT bInit AND stPositionState.bLocked THEN
        stCachedPositionState.sName := stPositionState.sName;
        stCachedPositionState.fPosition := stPositionState.fPosition;
        stCachedPositionState.fDelta := stPositionState.fDelta;
        stCachedPositionState.fVelocity := stPositionState.fVelocity;
        stCachedPositionState.fAccel := stPositionState.fAccel;
        stCachedPositionState.fDecel := stPositionState.fDecel;
        bInit := TRUE;
    // Do nothing, or unlock the state if bLocked goes FALSE
    ELSIF NOT stPositionState.bLocked THEN
        bInit := FALSE;
    END_IF
END_IF

END_FUNCTION_BLOCK

// POUs/Motion/States/FB_PositionStateMoveND

FUNCTION_BLOCK FB_PositionStateMoveND
(*
    This function block coordinates multidimensional state moves for groups of motors.
    It is a building block not meant for use outside of lcls-twintcat-motion.

    Use FB_PositionState1D, FB_PositionState2D, ... etc. instead
*)
VAR_IN_OUT
    // Array of motors to move together
    astMotionStage: ARRAY[1..MotionConstants.MAX_STATE_MOTORS] OF ST_MotionStage;
    // 1D Position states: the current position to send each axis to
    astPositionState: ARRAY[1..MotionConstants.MAX_STATE_MOTORS] OF ST_PositionState;
END_VAR
VAR_INPUT
    // The number of motors we're actually using
    nActiveMotorCount: UINT;
    // Start all moves on rising edge, stop all moves on falling edge
    bExecute: BOOL;
    // Reset any errors
    bReset: BOOL;
    // Define behavior for when a move request is interrupted with a new request
    enumMotionRequest: E_MotionRequest := E_MotionRequest.WAIT;
END_VAR
VAR_OUTPUT
    // TRUE if ALL of the motors are at their goal states
    bAtState: BOOL;
    // TRUE if ANY of this FB's moves are in progress
    bBusy: BOOL;
    // TRUE if ALL motors have completed the last move request from this FB
    bDone: BOOL;
    // TRUE if ANY of this FB's moves had an error
    bError: BOOL;
    // How many FBs are erroring
    nErrorCount: UINT;
    // Which component is the source of the example/summarized error
    nShownError: DINT;
    // One of the error ids
    nErrorID: UDINT;
    // The error error message matching the ID
    sErrorMessage: STRING;
END_VAR
VAR
    // 1D State movers: FBs to move the motors
    afbPositionStateMove: ARRAY[1..MotionConstants.MAX_STATE_MOTORS] OF FB_PositionStateMove;
    nIndex: DINT;
    bMotorCountError: BOOL;
    nLowerBound: DINT;
    nUpperBound: DINT;
END_VAR


CheckCount();
IF NOT bMotorCountError THEN
    DoStateMoves();
    CombineOutputs();
END_IF

ACTION CheckCount:

// Make sure the motor count is valid (positive, nonzero, less or equal to the max)
bMotorCountError S= nActiveMotorCount <= 0;
bMotorCountError S= nActiveMotorCount > MotionConstants.MAX_STATE_MOTORS;

IF bMotorCountError THEN
    bError := TRUE;
    sErrorMessage := 'Internal Error: invalid motor count';
END_IF
END_ACTION

ACTION CombineOutputs:

// bAtState is TRUE if ALL entries are TRUE
bAtState := TRUE;
FOR nIndex := 1 TO nActiveMotorCount DO
    bAtState := bAtState AND afbPositionStateMove[nIndex].bAtState;
END_FOR

// bBusy is TRUE if ANY entry is TRUE
bBusy := FALSE;
FOR nIndex := 1 TO nActiveMotorCount DO
    bBusy := bBusy OR afbPositionStateMove[nIndex].bBusy;
END_FOR

// bDone is TRUE if ALL entries are TRUE
bDone := TRUE;
FOR nIndex := 1 TO nActiveMotorCount DO
    bDone := bDone AND afbPositionStateMove[nIndex].bDone;
END_FOR

// bError is TRUE if ANY entry is TRUE
// also set nShownError and increment nErrorCount
bError := FALSE;
nErrorCount := 0;
FOR nIndex := 1 TO nActiveMotorCount DO
    bError := bError OR afbPositionStateMove[nIndex].bError;
    IF afbPositionStateMove[nIndex].bError THEN
        nShownError := nIndex;
        nErrorCount := nErrorCount + 1;
    END_IF
END_FOR

// Pick error id and message using nShownError
IF bError THEN
    nErrorID := afbPositionStateMove[nShownError].nErrorID;
    sErrorMessage := afbPositionStateMove[nShownError].sErrorMessage;
ELSE
    nErrorID := 0;
    sErrorMessage := '';
END_IF
END_ACTION

ACTION DoStateMoves:

// Do the individual moves
FOR nIndex := 1 TO nActiveMotorCount DO
    afbPositionStateMove[nIndex](
        stMotionStage:=astMotionStage[nIndex],
        stPositionState:=astPositionState[nIndex],
        bExecute:=bExecute,
        bReset:=bReset,
        enumMotionRequest:=enumMotionRequest,
    );
END_FOR
END_ACTION

END_FUNCTION_BLOCK

// POUs/Motion/States/FB_PositionStateMove
FUNCTION_BLOCK FB_PositionStateMove
(*
    Request a move to a particular state from an axis controlled via EPICS
    pytmc PVs here only exposed if using directly and not through another states function block.
*)
VAR_IN_OUT
    // Motor to move
    stMotionStage: ST_MotionStage;

    // State to move to
    {attribute 'pytmc' := '
        pv:
    '}
    stPositionState: ST_PositionState;
END_VAR
VAR_INPUT
    // Start move on rising edge, stop move on falling edge
    {attribute 'pytmc' := '
        pv: GO
        io: io
        field: ZNAM False
        field: ONAM True
    '}
    bExecute: BOOL;

    // Rising edge error reset
    {attribute 'pytmc' := '
        pv: RESET
        io: io
        field: ZNAM False
        field: ONAM True
    '}
    bReset: BOOL;

    // Define behavior for when a move is already active
    enumMotionRequest: E_MotionRequest := E_MotionRequest.WAIT;
END_VAR
VAR_OUTPUT
    // TRUE if the motor is at this state
    {attribute 'pytmc' := '
        pv: AT_STATE
        io: input
        field: ZNAM False
        field: ONAM True
    '}
    bAtState: BOOL;

    // TRUE if we have an error
    {attribute 'pytmc' := '
        pv: ERR
        io: input
        field: ZNAM False
        field: ONAM True
    '}
    bError: BOOL;

    // Error code
    {attribute 'pytmc' := '
        pv: ERRID
        io: input
    '}
    nErrorID: UDINT;

    // Error description
    {attribute 'pytmc' := '
        pv: ERRMSG
        io: input
    '}
    sErrorMessage: STRING;

    // TRUE if we are moving to a state
    {attribute 'pytmc' := '
        pv: BUSY
        io: input
        field: ZNAM False
        field: ONAM True
    '}
    bBusy: BOOL;

    // TRUE if we are not moving and we reached a state successfully on our last move
    {attribute 'pytmc' := '
        pv: DONE
        io: input
        field: ZNAM False
        field: ONAM True
    '}
    bDone: BOOL;
END_VAR
VAR
    fbMotionRequest: FB_MotionRequest;
    bAllowMove: BOOL;
END_VAR

// Veto the move for uninitialized and unsafe states
bAllowMove := stPositionState.bMoveOk AND stPositionState.bValid AND stPositionState.bUpdated;

// Do the move
fbMotionRequest(
    stMotionStage := stMotionStage,
    bExecute := bExecute AND bAllowMove,
    bReset := bReset,
    enumMotionRequest := enumMotionRequest,
    fPos := stPositionState.fPosition,
    fVel := stPositionState.fVelocity,
    fAcc := stPositionState.fAccel,
    fDec := stPositionState.fDecel,
    bError => bError,
    nErrorId => nErrorId,
    sErrorMessage => sErrorMessage,
    bBusy => bBusy,
    bDone => bDone);

// Inject custom error if we can't move because of bMoveOk or bValid
IF bExecute AND NOT bAllowMove THEN
    bError := TRUE;
    IF stPositionState.bValid THEN
        nErrorId := 16#7901;
    ELSE
        nErrorId := 16#7902;
    END_IF
    sErrorMessage := F_MotionErrorCodeLookup(nErrorId := nErrorID);
END_IF

// This can be useful if we're running this FB standalone for some reason
bAtState := F_AtPositionState(stMotionStage:=stMotionStage, stPositionState:=stPositionState);

END_FUNCTION_BLOCK

// POUs/Motion/States/Helpers/F_AtPositionState
FUNCTION F_AtPositionState : BOOL
(*
    Check if the motor is within the state bounds
    This will only run properly if FB_PositionStateInternal has been called on the position state to initialize it.
*)
VAR_INPUT
    stMotionStage: ST_MotionStage;
    stPositionState: ST_PositionState;
END_VAR

// If state is defined, we are within the delta, and we are either not moving or our destination is within the delta, we are at the state
F_AtPositionState := stPositionState.bValid AND stPositionState.bUpdated
                     AND F_PosWithinDelta(stMotionStage.stAxisStatus.fActPosition, stPositionState)
                     AND ((NOT stMotionStage.bExecute) OR F_PosWithinDelta(stMotionStage.fPosition, stPositionState));

END_FUNCTION

// POUs/Motion/States/Helpers/F_PosWithinDelta
FUNCTION F_PosWithinDelta : BOOL
VAR_INPUT
    fPosition: LREAL;
    stPositionState: ST_PositionState;
END_VAR

F_PosWithinDelta := F_PosOverLowerBound(fPosition, stPositionState) AND
                    F_PosUnderUpperBound(fPosition, stPositionState);

END_FUNCTION

// POUs/Motion/States/Helpers/F_PosOverLowerBound
FUNCTION F_PosOverLowerBound : BOOL
VAR_INPUT
    fPosition: LREAL;
    stPositionState: ST_PositionState;
END_VAR

F_PosOverLowerBound := fPosition > (stPositionState.fPosition - ABS(stPositionState.fDelta));

END_FUNCTION

// POUs/Motion/States/Helpers/F_PosUnderUpperBound
FUNCTION F_PosUnderUpperBound : BOOL
VAR_INPUT
    fPosition: LREAL;
    stPositionState: ST_PositionState;
END_VAR

F_PosUnderUpperBound := fPosition < (stPositionState.fPosition + ABS(stPositionState.fDelta));

END_FUNCTION

// POUs/Motion/FB_MotionRequest
FUNCTION_BLOCK FB_MotionRequest
(*
    Request a move from an axis controlled via EPICS using FB_MotionStage
    This exists to manage situations where different bits of code may need to move the same motor.
    With just the ST_MotionStage/FB_MotionStage setup it is possible for two function blocks to
    fight with and interfere with each other and with the EPICS commands.
*)
VAR_IN_OUT
    // Motor to move
    stMotionStage: ST_MotionStage;
END_VAR
VAR_INPUT
    // Start move on rising edge, stop move on falling edge
    bExecute: BOOL;
    // Reset errors on rising edge
    bReset: BOOL;
    // Define behavior for when the motor is already moving
    enumMotionRequest: E_MotionRequest := E_MotionRequest.WAIT;
    // Goal position
    fPos: LREAL;
    // Move velocity
    fVel: LREAL;
    // Optional acceleration
    fAcc: LREAL;
    // Optional deceleration
    fDec: LREAL;
END_VAR
VAR_OUTPUT
    // True if in error state
    bError: BOOL;
    // Error code
    nErrorId: UDINT;
    // What the error code means
    sErrorMessage: STRING;
    // If TRUE, we are moving the motor
    bBusy: BOOL;
    // If TRUE, we are not moving the motor and our most recent move was successful
    bDone: BOOL;
END_VAR
VAR
    rtExec: R_TRIG;
    ftExec: F_TRIG;
    rtReset: R_TRIG;
    ftBusy: F_TRIG;
    nState: UINT := 0;
    bMyMove: BOOL;
    bCausedError: BOOL;
END_VAR
// Define local constants for our state machine states
VAR CONSTANT
    INIT: UINT := 0;
    WAIT_EXEC: UINT := 1;
    PICK_REQUEST: UINT := 2;
    WAIT_OTHER_MOVE: UINT := 3;
    STOP_OTHER_MOVE: UINT := 4;
    START_MOVE: UINT := 5;
    WAIT_MY_MOVE: UINT := 6;
    STOP_MY_MOVE: UINT := 7;
    DONE_MOVING: UINT := 8;
    ERROR: UINT := 9;
END_VAR

rtExec(CLK:=bExecute);
ftExec(CLK:=bExecute);
rtReset(CLK:=bReset);

// Go back to INIT state on reset
IF rtReset.Q THEN
    nState := INIT;
    stMotionStage.bReset := TRUE;
END_IF
IF rtExec.Q OR ftExec.Q THEN
    bDone := FALSE;
END_IF

CASE nState OF
    // Start by setting everything to a known value
    INIT:
        nState := WAIT_EXEC;
        bError := FALSE;
        sErrorMessage := '';
        bDone := FALSE;
        bCausedError := FALSE;
    // Normal "waiting for move command" state
    WAIT_EXEC:
        bMyMove := FALSE;
        // Looking for a rising edge on bExecute
        IF rtExec.Q THEN
            bDone := FALSE;
            nState := PICK_REQUEST;
        END_IF
    // Decide how to handle the request
    PICK_REQUEST:
        IF stMotionStage.bBusy THEN
            CASE enumMotionRequest OF
                E_MotionRequest.WAIT:
                    nState := WAIT_OTHER_MOVE;
                E_MotionRequest.INTERRUPT:
                    nState := STOP_OTHER_MOVE;
                E_MotionRequest.ABORT:
                    nState := ERROR;
                    bError := TRUE;
                    nErrorId := 16#7900;
            END_CASE
        ELSE
            nState := START_MOVE;
        END_IF
    // Watch the other move, then see if it's our turn
    WAIT_OTHER_MOVE:
        IF NOT stMotionStage.bBusy THEN
            // Try to pick request again next cycle once the move is over
            nState := PICK_REQUEST;
        END_IF
    // Interrupt the other move, then go to start ours
    STOP_OTHER_MOVE:
        stMotionStage.bExecute := FALSE;
        IF NOT stMotionStage.bBusy THEN
            nState := START_MOVE;
        END_IF
    // Set the correct values on ST_MotionStage to start a new absolute move
    START_MOVE:
        bMyMove := TRUE;
        stMotionStage.bExecute := TRUE;
        stMotionStage.nCommand := E_EpicsMotorCmd.MOVE_ABSOLUTE;
        stMotionStage.fPosition := fPos;
        stMotionStage.fVelocity := fVel;
        stMotionStage.fAcceleration := fAcc;
        stMotionStage.fDeceleration := fDec;
        nState := WAIT_MY_MOVE;
    // Watch our ongoing move, look for the move to end or requests to stop the move from this FB
    WAIT_MY_MOVE:
        ftBusy(CLK:=stMotionStage.bBusy);
        IF ftBusy.Q THEN
            nState := DONE_MOVING;
        END_IF
        // Implement stop on falling trigger
        IF ftExec.Q THEN
            nState := STOP_MY_MOVE;
        END_IF
    // Request a stop and wait for it to happen
    STOP_MY_MOVE:
        stMotionStage.bExecute := FALSE;
        IF NOT stMotionStage.bBusy THEN
            nState := DONE_MOVING;
        END_IF
    // Pick out the bDone state and return to waiting
    DONE_MOVING:
        bDone := stMotionStage.bDone;
        nState := WAIT_EXEC;
    // Lock us into the error state until the FB is reset
    ERROR:
        bMyMove := FALSE;
END_CASE

// Transition to the ERROR state if applicable
IF bMyMove AND stMotionStage.bError THEN
    nState := ERROR;
    bError := TRUE;
    nErrorId := stMotionStage.nErrorId;
    bCausedError := TRUE;
END_IF
sErrorMessage := F_MotionErrorCodeLookup(nErrorId := nErrorId);

CASE nState OF
INIT, WAIT_EXEC, ERROR:
    bBusy := FALSE;
ELSE
    bBusy := TRUE;
END_CASE

END_FUNCTION_BLOCK

// POUs/Motion/States/FB_PositionStateReadND
FUNCTION_BLOCK FB_PositionStateReadND
(*
    Function block to get the combined N-dimensional state of a group of motors.
    It is a building block not meant for use outside of lcls-twintcat-motion.

    Use FB_PositionStateRead1D, FB_PositionStateRead2D, ... etc. instead
*)
VAR_IN_OUT
    // The motors with a combined N-dimensional state
    astMotionStage: ARRAY[1..MotionConstants.MAX_STATE_MOTORS] OF ST_MotionStage;
    // Each motor's respective position states along its direction
    astPositionState: ARRAY[1..MotionConstants.MAX_STATE_MOTORS] OF ARRAY[1..GeneralConstants.MAX_STATES] OF ST_PositionState;
END_VAR
VAR_INPUT
    // The number of motors we're actually using
    nActiveMotorCount: UINT;
END_VAR
VAR_OUTPUT
    // TRUE if we're standing still at a known state.
    bKnownState: BOOL;
    // TRUE if we're moving, there can be no valid state if we are moving.
    bMovingState: BOOL;
    // If we're at a known state, this will be the state index along the enclosed states arrays. Otherwise, it will be zero, which is below the bounds of the states array.
    nPositionIndex: UINT;
    // TRUE if the active motor count was invalid
    bMotorCountError: BOOL;
    // A full description of whether we're at each of our states. This is used to clarify cases where states may overlap.
    abAtPosition: ARRAY[1..GeneralConstants.MAX_STATES] OF BOOL;
END_VAR
VAR
    // The individual position state reader function blocks
    afbPositionStateRead: ARRAY[1..MotionConstants.MAX_STATE_MOTORS] OF FB_PositionStateRead;

    nIter: UINT;
    nIter2: UINT;
END_VAR


CheckCount();
IF NOT bMotorCountError THEN
    DoStateReads();
    CombineOutputs();
END_IF

ACTION CheckCount:

// Make sure the motor count is valid (positive, nonzero, less or equal to the max)
bMotorCountError S= nActiveMotorCount <= 0;
bMotorCountError S= nActiveMotorCount > MotionConstants.MAX_STATE_MOTORS;
END_ACTION

ACTION CombineOutputs:

// bKnownState is TRUE if ALL motors have the same known state
bKnownState := TRUE;
FOR nIter := 1 TO nActiveMotorCount DO
    bKnownState := bKnownState AND afbPositionStateRead[nIter].bKnownState;
END_FOR

// bMovingState is TRUE if ANY motor is moving
bMovingState := FALSE;
FOR nIter := 1 TO nActiveMotorCount DO
    bMovingState := bMovingState OR afbPositionStateRead[nIter].bMovingState;
END_FOR

// To account for redundant 1D states, we need to check the full output arrays.
nPositionIndex := 0;
FOR nIter := 1 TO GeneralConstants.MAX_STATES DO
    abAtPosition[nIter] := TRUE;
    FOR nIter2 := 1 TO nActiveMotorCount DO
        abAtPosition[nIter] R= NOT afbPositionStateRead[nIter2].abAtPosition[nIter];
    END_FOR
    IF abAtPosition[nIter] THEN
        nPositionIndex := nIter;
    END_IF
END_FOR

// Position index 0 means different positions
bKnownState := bKnownState AND nPositionIndex <> 0;
END_ACTION

ACTION DoStateReads:

MOTION_GVL.nMaxStateMotorCount := MAX(MOTION_GVL.nMaxStateMotorCount, nActiveMotorCount);
FOR nIter := 1 TO nActiveMotorCount DO
    afbPositionStateRead[nIter](
        stMotionStage:=astMotionStage[nIter],
        astPositionState:=astPositionState[nIter],
    );
END_FOR
END_ACTION

END_FUNCTION_BLOCK

// POUs/Motion/States/FB_PositionStateRead
FUNCTION_BLOCK FB_PositionStateRead
(*
    This function block tells us what state a single motor is at.
    In the case of multiple valid overlapping states, one will be picked arbitrarily,
    but we can see a full description of which overlapping states are present using the abAtPosition array.

